LIN {X 0,Y 296.681,Z 512.231,A -85,B 0,C 180,E1 -16490.81,E2 -16490.81} C_VEL
LIN {X 0,Y 296.616,Z 512.901,A -85,B 0,C 180,E1 -16492.472,E2 -16492.472} C_VEL
LIN {X 0,Y 296.719,Z 512.686,A -85,B 0,C 180,E1 -16495.232,E2 -16495.232} C_VEL
LIN {X 0,Y 296.911,Z 511.914,A -85,B 0,C 180,E1 -16496.723,E2 -16496.723} C_VEL
LIN {X 0,Y 297.383,Z 509.725,A -85,B 0,C 180,E1 -16499.024,E2 -16499.024} C_VEL
LIN {X 0,Y 298.001,Z 506.45,A -85,B 0,C 180,E1 -16501.251,E2 -16501.251} C_VEL
LIN {X 0,Y 298.906,Z 501.771,A -85,B 0,C 180,E1 -16503.538,E2 -16503.538} C_VEL
LIN {X 0,Y 300.159,Z 495.578,A -85,B 0,C 180,E1 -16505.824,E2 -16505.824} C_VEL
LIN {X 0,Y 301.385,Z 489.056,A -85,B 0,C 180,E1 -16507.716,E2 -16507.716} C_VEL
LIN {X 0,Y 302.931,Z 480.785,A -85,B 0,C 180,E1 -16509.639,E2 -16509.639} C_VEL
LIN {X 0,Y 304.466,Z 471.668,A -85,B 0,C 180,E1 -16511.353,E2 -16511.353} C_VEL
LIN {X 0,Y 306.154,Z 461.176,A -85,B 0,C 180,E1 -16512.929,E2 -16512.929} C_VEL
LIN {X 0,Y 307.794,Z 449.247,A -85,B 0,C 180,E1 -16514.327,E2 -16514.327} C_VEL
LIN {X 0,Y 307.85,Z 445.631,A -85,B 0,C 180,E1 -16514.72,E2 -16514.72} C_VEL
LIN {X 0,Y 305.288,Z 433.549,A -85,B 0,C 180,E1 -16516.069,E2 -16516.069} C_VEL
LIN {X 0,Y 301.496,Z 421.211,A -85,B 0,C 180,E1 -16517.278,E2 -16517.278} C_VEL
LIN {X 0,Y 297.926,Z 411.655,A -85,B 0,C 180,E1 -16518.096,E2 -16518.096} C_VEL
LIN {X 0,Y 297.834,Z 411.063,A -85,B 0,C 180,E1 -16518.137,E2 -16518.137} C_VEL
LIN {X 0,Y 298.025,Z 408.055,A -85,B 0,C 180,E1 -16522.184,E2 -16522.184} C_VEL
LIN {X 0,Y 298.192,Z 405.628,A -85,B 0,C 180,E1 -16525.572,E2 -16525.572} C_VEL
LIN {X 0,Y 298.291,Z 403.444,A -85,B 0,C 180,E1 -16528.779,E2 -16528.779} C_VEL
LIN {X 0,Y 298.434,Z 403.312,A -85,B 0,C 180,E1 -16531.901,E2 -16531.901} C_VEL
LIN {X 0,Y 298.483,Z 403.308,A -85,B 0,C 180,E1 -16534.924,E2 -16534.924} C_VEL
LIN {X 0,Y 298.482,Z 403.306,A -85,B 0,C 180,E1 -16537.869,E2 -16537.869} C_VEL
LIN {X 0,Y 298.55,Z 403.298,A -85,B 0,C 180,E1 -16540.758,E2 -16540.758} C_VEL
LIN {X 0,Y 298.575,Z 403.294,A -85,B 0,C 180,E1 -16544.994,E2 -16544.994} C_VEL
LIN {X 0,Y 298.577,Z 403.292,A -85,B 0,C 180,E1 -16549.146,E2 -16549.146} C_VEL
LIN {X 0,Y 298.735,Z 403.271,A -85,B 0,C 180,E1 -16552.197,E2 -16552.197} C_VEL
LIN {X 0,Y 298.066,Z 403.353,A -85,B 0,C 180,E1 -16553.321,E2 -16553.321} C_VEL
LIN {X 0,Y 295.213,Z 403.713,A -85,B 0,C 180,E1 -16555.151,E2 -16555.151} C_VEL
LIN {X 0,Y 292.833,Z 404.01,A -85,B 0,C 180,E1 -16556.636,E2 -16556.636} C_VEL
LIN {X 0,Y 291.871,Z 404.129,A -85,B 0,C 180,E1 -16557.787,E2 -16557.787} C_VEL
LIN {X 0,Y 291.823,Z 404.132,A -85,B 0,C 180,E1 -16558.176,E2 -16558.176} C_VEL
LIN {X 0,Y 291.962,Z 404.118,A -85,B 0,C 180,E1 -16560,E2 -16560} C_VEL
LIN {X 0,Y 291.788,Z 404.139,A -85,B 0,C 180,E1 -16562.761,E2 -16562.761} C_VEL
LIN {X 0,Y 291.727,Z 404.147,A -85,B 0,C 180,E1 -16566.918,E2 -16566.918} C_VEL
LIN {X 0,Y 291.611,Z 404.161,A -85,B 0,C 180,E1 -16569.713,E2 -16569.713} C_VEL
LIN {X 0,Y 291.505,Z 404.175,A -85,B 0,C 180,E1 -16573.951,E2 -16573.951} C_VEL
LIN {X 0,Y 291.471,Z 404.181,A -85,B 0,C 180,E1 -16576.819,E2 -16576.819} C_VEL
LIN {X 0,Y 291.479,Z 404.18,A -85,B 0,C 180,E1 -16579.901,E2 -16579.901} C_VEL
LIN {X 0,Y 291.422,Z 404.189,A -85,B 0,C 180,E1 -16584.204,E2 -16584.204} C_VEL
LIN {X 0,Y 291.404,Z 404.192,A -85,B 0,C 180,E1 -16587.274,E2 -16587.274} C_VEL
LIN {X 0,Y 291.319,Z 404.202,A -85,B 0,C 180,E1 -16590.439,E2 -16590.439} C_VEL
LIN {X 0,Y 291.33,Z 404.198,A -85,B 0,C 180,E1 -16593.701,E2 -16593.701} C_VEL
LIN {X 0,Y 291.43,Z 404.372,A -85,B 0,C 180,E1 -16597.077,E2 -16597.077} C_VEL
LIN {X 0,Y 292.013,Z 407.676,A -85,B 0,C 180,E1 -16600.528,E2 -16600.528} C_VEL
LIN {X 0,Y 292.688,Z 411.501,A -85,B 0,C 180,E1 -16604.135,E2 -16604.135} C_VEL
LIN {X 0,Y 293.487,Z 415.946,A -85,B 0,C 180,E1 -16607.932,E2 -16607.932} C_VEL
LIN {X 0,Y 294.295,Z 420.631,A -85,B 0,C 180,E1 -16611.622,E2 -16611.622} C_VEL
LIN {X 0,Y 294.316,Z 423.007,A -85,B 0,C 180,E1 -16613.35,E2 -16613.35} C_VEL
LIN {X 0,Y 293.501,Z 427.798,A -85,B 0,C 180,E1 -16616.586,E2 -16616.586} C_VEL
LIN {X 0,Y 292.428,Z 433.947,A -85,B 0,C 180,E1 -16620.555,E2 -16620.555} C_VEL
LIN {X 0,Y 291.578,Z 439.819,A -85,B 0,C 180,E1 -16624.22,E2 -16624.22} C_VEL
LIN {X 0,Y 294.842,Z 453.988,A -85,B 0,C 180,E1 -16625.215,E2 -16625.215} C_VEL
LIN {X 0,Y 296.937,Z 466.347,A -85,B 0,C 180,E1 -16626.278,E2 -16626.278} C_VEL
LIN {X 0,Y 297.877,Z 477.919,A -85,B 0,C 180,E1 -16627.433,E2 -16627.433} C_VEL
LIN {X 0,Y 298.271,Z 489.026,A -85,B 0,C 180,E1 -16628.763,E2 -16628.763} C_VEL
LIN {X 0,Y 298.073,Z 493.023,A -85,B 0,C 180,E1 -16629.291,E2 -16629.291} C_VEL
LIN {X 0,Y 296.243,Z 503.418,A -85,B 0,C 180,E1 -16630.785,E2 -16630.785} C_VEL
LIN {X 0,Y 294.557,Z 512.927,A -85,B 0,C 180,E1 -16632.496,E2 -16632.496} C_VEL
LIN {X 0,Y 293.442,Z 519.865,A -85,B 0,C 180,E1 -16634.016,E2 -16634.016} C_VEL
LIN {X 0,Y 292.007,Z 527.627,A -85,B 0,C 180,E1 -16636.076,E2 -16636.076} C_VEL
LIN {X 0,Y 290.904,Z 533.892,A -85,B 0,C 180,E1 -16638.153,E2 -16638.153} C_VEL
LIN {X 0,Y 290.221,Z 538.898,A -85,B 0,C 180,E1 -16640.243,E2 -16640.243} C_VEL
LIN {X 0,Y 289.814,Z 542.782,A -85,B 0,C 180,E1 -16642.338,E2 -16642.338} C_VEL
LIN {X 0,Y 289.624,Z 545.643,A -85,B 0,C 180,E1 -16644.433,E2 -16644.433} C_VEL
LIN {X 0,Y 289.583,Z 547.008,A -85,B 0,C 180,E1 -16645.827,E2 -16645.827} C_VEL
LIN {X 0,Y 289.557,Z 547.975,A -85,B 0,C 180,E1 -16647.22,E2 -16647.22} C_VEL
LIN {X 0,Y 289.58,Z 548.533,A -85,B 0,C 180,E1 -16648.612,E2 -16648.612} C_VEL
LIN {X 0,Y 289.694,Z 548.659,A -85,B 0,C 180,E1 -16650.003,E2 -16650.003} C_VEL
LIN {X 0,Y 289.609,Z 548.378,A -85,B 0,C 180,E1 -16651.393,E2 -16651.393} C_VEL
LIN {X 0,Y 289.567,Z 547.706,A -85,B 0,C 180,E1 -16652.785,E2 -16652.785} C_VEL
LIN {X 0,Y 289.601,Z 546.628,A -85,B 0,C 180,E1 -16654.178,E2 -16654.178} C_VEL
LIN {X 0,Y 289.637,Z 544.779,A -85,B 0,C 180,E1 -16655.81,E2 -16655.81} C_VEL
LIN {X 0,Y 289.908,Z 540.719,A -85,B 0,C 180,E1 -16658.366,E2 -16658.366} C_VEL
LIN {X 0,Y 290.45,Z 536.166,A -85,B 0,C 180,E1 -16660.458,E2 -16660.458} C_VEL
LIN {X 0,Y 291.383,Z 529.252,A -85,B 0,C 180,E1 -16662.894,E2 -16662.894} C_VEL
LIN {X 0,Y 292.59,Z 521.762,A -85,B 0,C 180,E1 -16664.967,E2 -16664.967} C_VEL
LIN {X 0,Y 293.871,Z 514.132,A -85,B 0,C 180,E1 -16666.68,E2 -16666.68} C_VEL
LIN {X 0,Y 295.154,Z 504.871,A -85,B 0,C 180,E1 -16668.393,E2 -16668.393} C_VEL
LIN {X 0,Y 296.846,Z 494.612,A -85,B 0,C 180,E1 -16669.9,E2 -16669.9} C_VEL
LIN {X 0,Y 297.487,Z 489.241,A -85,B 0,C 180,E1 -16670.576,E2 -16670.576} C_VEL
LIN {X 0,Y 296.781,Z 477.347,A -85,B 0,C 180,E1 -16671.956,E2 -16671.956} C_VEL
LIN {X 0,Y 295.703,Z 465.945,A -85,B 0,C 180,E1 -16673.033,E2 -16673.033} C_VEL
LIN {X 0,Y 293.736,Z 453.233,A -85,B 0,C 180,E1 -16674.003,E2 -16674.003} C_VEL
LIN {X 0,Y 291.321,Z 441.044,A -85,B 0,C 180,E1 -16674.724,E2 -16674.724} C_VEL
LIN {X 0,Y 292.187,Z 434.465,A -85,B 0,C 180,E1 -16678.757,E2 -16678.757} C_VEL
LIN {X 0,Y 293.285,Z 427.694,A -85,B 0,C 180,E1 -16682.996,E2 -16682.996} C_VEL
LIN {X 0,Y 294.052,Z 423.605,A -85,B 0,C 180,E1 -16685.647,E2 -16685.647} C_VEL
LIN {X 0,Y 294.158,Z 420.178,A -85,B 0,C 180,E1 -16687.96,E2 -16687.96} C_VEL
LIN {X 0,Y 293.255,Z 414.608,A -85,B 0,C 180,E1 -16692.018,E2 -16692.018} C_VEL
LIN {X 0,Y 292.387,Z 409.776,A -85,B 0,C 180,E1 -16695.808,E2 -16695.808} C_VEL
LIN {X 0,Y 291.492,Z 404.752,A -85,B 0,C 180,E1 -16700.024,E2 -16700.024} C_VEL
LIN {X 0,Y 291.369,Z 404.193,A -85,B 0,C 180,E1 -16700.524,E2 -16700.524} C_VEL
LIN {X 0,Y 291.415,Z 404.187,A -85,B 0,C 180,E1 -16702.92,E2 -16702.92} C_VEL
LIN {X 0,Y 291.352,Z 404.194,A -85,B 0,C 180,E1 -16706.302,E2 -16706.302} C_VEL
LIN {X 0,Y 291.391,Z 404.189,A -85,B 0,C 180,E1 -16710.262,E2 -16710.262} C_VEL
LIN {X 0,Y 291.42,Z 404.185,A -85,B 0,C 180,E1 -16714.272,E2 -16714.272} C_VEL
LIN {X 0,Y 291.389,Z 404.186,A -85,B 0,C 180,E1 -16717.3,E2 -16717.3} C_VEL
LIN {X 0,Y 291.466,Z 404.181,A -85,B 0,C 180,E1 -16720.271,E2 -16720.271} C_VEL
LIN {X 0,Y 291.549,Z 404.171,A -85,B 0,C 180,E1 -16724.635,E2 -16724.635} C_VEL
LIN {X 0,Y 291.543,Z 404.169,A -85,B 0,C 180,E1 -16728.881,E2 -16728.881} C_VEL
LIN {X 0,Y 291.695,Z 404.15,A -85,B 0,C 180,E1 -16731.688,E2 -16731.688} C_VEL
LIN {X 0,Y 291.632,Z 404.159,A -85,B 0,C 180,E1 -16734.468,E2 -16734.468} C_VEL
LIN {X 0,Y 291.895,Z 404.124,A -85,B 0,C 180,E1 -16738.62,E2 -16738.62} C_VEL
LIN {X 0,Y 291.895,Z 404.123,A -85,B 0,C 180,E1 -16741.38,E2 -16741.38} C_VEL
LIN {X 0,Y 291.753,Z 404.129,A -85,B 0,C 180,E1 -16746.918,E2 -16746.918} C_VEL
LIN {X 0,Y 291.637,Z 404.153,A -85,B 0,C 180,E1 -16749.712,E2 -16749.712} C_VEL
LIN {X 0,Y 291.529,Z 404.172,A -85,B 0,C 180,E1 -16753.95,E2 -16753.95} C_VEL
LIN {X 0,Y 291.494,Z 404.17,A -85,B 0,C 180,E1 -16756.817,E2 -16756.817} C_VEL
LIN {X 0,Y 291.459,Z 404.17,A -85,B 0,C 180,E1 -16759.874,E2 -16759.874} C_VEL
LIN {X 0,Y 291.408,Z 404.183,A -85,B 0,C 180,E1 -16764.205,E2 -16764.205} C_VEL
LIN {X 0,Y 291.427,Z 404.184,A -85,B 0,C 180,E1 -16767.271,E2 -16767.271} C_VEL
LIN {X 0,Y 291.341,Z 404.188,A -85,B 0,C 180,E1 -16770.436,E2 -16770.436} C_VEL
LIN {X 0,Y 291.351,Z 404.188,A -85,B 0,C 180,E1 -16773.697,E2 -16773.697} C_VEL
LIN {X 0,Y 291.379,Z 404.19,A -85,B 0,C 180,E1 -16777.252,E2 -16777.252} C_VEL
LIN {X 0,Y 291.34,Z 404.192,A -85,B 0,C 180,E1 -16780.641,E2 -16780.641} C_VEL
LIN {X 0,Y 291.32,Z 404.188,A -85,B 0,C 180,E1 -16784.396,E2 -16784.396} C_VEL
LIN {X 0,Y 291.333,Z 404.193,A -85,B 0,C 180,E1 -16788.403,E2 -16788.403} C_VEL
LIN {X 0,Y 291.354,Z 404.19,A -85,B 0,C 180,E1 -16791.156,E2 -16791.156} C_VEL
LIN {X 0,Y 291.367,Z 404.189,A -85,B 0,C 180,E1 -16794.624,E2 -16794.624} C_VEL
LIN {X 0,Y 291.376,Z 404.188,A -85,B 0,C 180,E1 -16797.949,E2 -16797.949} C_VEL
LIN {X 0,Y 291.383,Z 404.191,A -85,B 0,C 180,E1 -16801.156,E2 -16801.156} C_VEL
LIN {X 0,Y 291.418,Z 404.185,A -85,B 0,C 180,E1 -16804.27,E2 -16804.27} C_VEL
LIN {X 0,Y 291.387,Z 404.188,A -85,B 0,C 180,E1 -16807.298,E2 -16807.298} C_VEL
LIN {X 0,Y 291.463,Z 404.179,A -85,B 0,C 180,E1 -16810.268,E2 -16810.268} C_VEL
LIN {X 0,Y 291.544,Z 404.171,A -85,B 0,C 180,E1 -16814.632,E2 -16814.632} C_VEL
LIN {X 0,Y 291.413,Z 404.184,A -85,B 0,C 180,E1 -16817.462,E2 -16817.462} C_VEL
LIN {X 0,Y 291.24,Z 404.209,A -85,B 0,C 180,E1 -16820.273,E2 -16820.273} C_VEL
LIN {X 0,Y 291.175,Z 404.529,A -85,B 0,C 180,E1 -16821.731,E2 -16821.731} C_VEL
LIN {X 0,Y 291.222,Z 406.671,A -85,B 0,C 180,E1 -16824.458,E2 -16824.458} C_VEL
LIN {X 0,Y 290.562,Z 409.89,A -85,B 0,C 180,E1 -16828.438,E2 -16828.438} C_VEL
LIN {X 0,Y 294.972,Z 424.125,A -85,B 0,C 180,E1 -16829.537,E2 -16829.537} C_VEL
LIN {X 0,Y 297.721,Z 434.159,A -85,B 0,C 180,E1 -16830.483,E2 -16830.483} C_VEL
LIN {X 0,Y 299.896,Z 445.157,A -85,B 0,C 180,E1 -16831.676,E2 -16831.676} C_VEL
LIN {X 0,Y 298.681,Z 455.984,A -85,B 0,C 180,E1 -16832.863,E2 -16832.863} C_VEL
LIN {X 0,Y 297.212,Z 466.632,A -85,B 0,C 180,E1 -16834.335,E2 -16834.335} C_VEL
LIN {X 0,Y 295.569,Z 477.057,A -85,B 0,C 180,E1 -16836.14,E2 -16836.14} C_VEL
LIN {X 0,Y 294.202,Z 485.218,A -85,B 0,C 180,E1 -16837.892,E2 -16837.892} C_VEL
LIN {X 0,Y 293.014,Z 491.971,A -85,B 0,C 180,E1 -16839.663,E2 -16839.663} C_VEL
LIN {X 0,Y 291.926,Z 498.542,A -85,B 0,C 180,E1 -16841.805,E2 -16841.805} C_VEL
LIN {X 0,Y 291.052,Z 503.752,A -85,B 0,C 180,E1 -16843.97,E2 -16843.97} C_VEL
LIN {X 0,Y 290.419,Z 507.763,A -85,B 0,C 180,E1 -16846.155,E2 -16846.155} C_VEL
LIN {X 0,Y 289.832,Z 511.314,A -85,B 0,C 180,E1 -16848.969,E2 -16848.969} C_VEL
LIN {X 0,Y 289.554,Z 512.957,A -85,B 0,C 180,E1 -16851.347,E2 -16851.347} C_VEL
LIN {X 0,Y 289.519,Z 513.386,A -85,B 0,C 180,E1 -16852.851,E2 -16852.851} C_VEL
LIN {X 0,Y 289.572,Z 513.384,A -85,B 0,C 180,E1 -16854.364,E2 -16854.364} C_VEL
LIN {X 0,Y 289.755,Z 512.734,A -85,B 0,C 180,E1 -16856.177,E2 -16856.177} C_VEL
LIN {X 0,Y 290.291,Z 510.467,A -85,B 0,C 180,E1 -16858.957,E2 -16858.957} C_VEL
LIN {X 0,Y 290.957,Z 507.246,A -85,B 0,C 180,E1 -16861.283,E2 -16861.283} C_VEL
LIN {X 0,Y 291.87,Z 502.682,A -85,B 0,C 180,E1 -16863.626,E2 -16863.626} C_VEL
LIN {X 0,Y 293.114,Z 496.848,A -85,B 0,C 180,E1 -16865.886,E2 -16865.886} C_VEL
LIN {X 0,Y 294.559,Z 489.677,A -85,B 0,C 180,E1 -16868.061,E2 -16868.061} C_VEL
LIN {X 0,Y 296.268,Z 480.874,A -85,B 0,C 180,E1 -16870.146,E2 -16870.146} C_VEL
LIN {X 0,Y 298.012,Z 471.092,A -85,B 0,C 180,E1 -16871.998,E2 -16871.998} C_VEL
LIN {X 0,Y 299.664,Z 461.06,A -85,B 0,C 180,E1 -16873.502,E2 -16873.502} C_VEL
LIN {X 0,Y 301.294,Z 449.764,A -85,B 0,C 180,E1 -16874.846,E2 -16874.846} C_VEL
LIN {X 0,Y 301.051,Z 445.998,A -85,B 0,C 180,E1 -16875.293,E2 -16875.293} C_VEL
LIN {X 0,Y 298.548,Z 434.444,A -85,B 0,C 180,E1 -16876.638,E2 -16876.638} C_VEL
LIN {X 0,Y 294.976,Z 422.795,A -85,B 0,C 180,E1 -16877.84,E2 -16877.84} C_VEL
LIN {X 0,Y 290.933,Z 412.057,A -85,B 0,C 180,E1 -16878.81,E2 -16878.81} C_VEL
LIN {X 0,Y 290.844,Z 411.521,A -85,B 0,C 180,E1 -16878.875,E2 -16878.875} C_VEL
LIN {X 0,Y 291.05,Z 408.634,A -85,B 0,C 180,E1 -16882.866,E2 -16882.866} C_VEL
LIN {X 0,Y 291.196,Z 406.275,A -85,B 0,C 180,E1 -16886.282,E2 -16886.282} C_VEL
LIN {X 0,Y 291.268,Z 404.208,A -85,B 0,C 180,E1 -16889.555,E2 -16889.555} C_VEL
LIN {X 0,Y 291.423,Z 404.186,A -85,B 0,C 180,E1 -16893.155,E2 -16893.155} C_VEL
LIN {X 0,Y 291.436,Z 404.186,A -85,B 0,C 180,E1 -16897.304,E2 -16897.304} C_VEL
LIN {X 0,Y 291.497,Z 404.175,A -85,B 0,C 180,E1 -16900.273,E2 -16900.273} C_VEL
LIN {X 0,Y 291.522,Z 404.17,A -85,B 0,C 180,E1 -16904.634,E2 -16904.634} C_VEL
LIN {X 0,Y 291.52,Z 404.172,A -85,B 0,C 180,E1 -16908.88,E2 -16908.88} C_VEL
LIN {X 0,Y 291.685,Z 404.148,A -85,B 0,C 180,E1 -16912.201,E2 -16912.201} C_VEL
LIN {X 0,Y 291.773,Z 404.141,A -85,B 0,C 180,E1 -16917.239,E2 -16917.239} C_VEL
LIN {X 0,Y 291.823,Z 404.132,A -85,B 0,C 180,E1 -16918.176,E2 -16918.176} C_VEL
LIN {X 0,Y 291.206,Z 404.212,A -85,B 0,C 180,E1 -16919.329,E2 -16919.329} C_VEL
LIN {X 0,Y 288.248,Z 404.587,A -85,B 0,C 180,E1 -16921.201,E2 -16921.201} C_VEL
LIN {X 0,Y 285.69,Z 404.905,A -85,B 0,C 180,E1 -16922.722,E2 -16922.722} C_VEL
LIN {X 0,Y 284.59,Z 405.037,A -85,B 0,C 180,E1 -16923.904,E2 -16923.904} C_VEL
LIN {X 0,Y 284.504,Z 405.045,A -85,B 0,C 180,E1 -16924.305,E2 -16924.305} C_VEL
LIN {X 0,Y 284.679,Z 405.025,A -85,B 0,C 180,E1 -16927.091,E2 -16927.091} C_VEL
LIN {X 0,Y 284.549,Z 405.042,A -85,B 0,C 180,E1 -16929.956,E2 -16929.956} C_VEL
LIN {X 0,Y 284.464,Z 405.052,A -85,B 0,C 180,E1 -16934.304,E2 -16934.304} C_VEL
LIN {X 0,Y 284.412,Z 405.058,A -85,B 0,C 180,E1 -16937.249,E2 -16937.249} C_VEL
LIN {X 0,Y 284.411,Z 405.059,A -85,B 0,C 180,E1 -16940.24,E2 -16940.24} C_VEL
LIN {X 0,Y 284.385,Z 405.066,A -85,B 0,C 180,E1 -16943.891,E2 -16943.891} C_VEL
LIN {X 0,Y 284.313,Z 405.076,A -85,B 0,C 180,E1 -16948.013,E2 -16948.013} C_VEL
LIN {X 0,Y 284.278,Z 405.078,A -85,B 0,C 180,E1 -16951.277,E2 -16951.277} C_VEL
LIN {X 0,Y 284.334,Z 405.068,A -85,B 0,C 180,E1 -16955.805,E2 -16955.805} C_VEL
LIN {X 0,Y 284.653,Z 406.913,A -85,B 0,C 180,E1 -16958.115,E2 -16958.115} C_VEL
LIN {X 0,Y 285.281,Z 410.368,A -85,B 0,C 180,E1 -16961.695,E2 -16961.695} C_VEL
LIN {X 0,Y 285.991,Z 414.396,A -85,B 0,C 180,E1 -16965.451,E2 -16965.451} C_VEL
LIN {X 0,Y 286.83,Z 419.085,A -85,B 0,C 180,E1 -16969.427,E2 -16969.427} C_VEL
LIN {X 0,Y 287.326,Z 422.758,A -85,B 0,C 180,E1 -16972.306,E2 -16972.306} C_VEL
LIN {X 0,Y 286.95,Z 426.313,A -85,B 0,C 180,E1 -16974.865,E2 -16974.865} C_VEL
LIN {X 0,Y 285.649,Z 433.115,A -85,B 0,C 180,E1 -16979.444,E2 -16979.444} C_VEL
LIN {X 0,Y 284.685,Z 439.351,A -85,B 0,C 180,E1 -16983.471,E2 -16983.471} C_VEL
LIN {X 0,Y 287.348,Z 450.529,A -85,B 0,C 180,E1 -16984.276,E2 -16984.276} C_VEL
LIN {X 0,Y 289.767,Z 463.231,A -85,B 0,C 180,E1 -16985.37,E2 -16985.37} C_VEL
LIN {X 0,Y 291.055,Z 475.183,A -85,B 0,C 180,E1 -16986.574,E2 -16986.574} C_VEL
LIN {X 0,Y 291.496,Z 487.557,A -85,B 0,C 180,E1 -16988.059,E2 -16988.059} C_VEL
LIN {X 0,Y 291.227,Z 494.231,A -85,B 0,C 180,E1 -16988.966,E2 -16988.966} C_VEL
LIN {X 0,Y 289.334,Z 504.284,A -85,B 0,C 180,E1 -16990.492,E2 -16990.492} C_VEL
LIN {X 0,Y 287.645,Z 513.364,A -85,B 0,C 180,E1 -16992.208,E2 -16992.208} C_VEL
LIN {X 0,Y 286.302,Z 520.998,A -85,B 0,C 180,E1 -16993.972,E2 -16993.972} C_VEL
LIN {X 0,Y 284.863,Z 528.465,A -85,B 0,C 180,E1 -16996.084,E2 -16996.084} C_VEL
LIN {X 0,Y 283.668,Z 535.378,A -85,B 0,C 180,E1 -16998.571,E2 -16998.571} C_VEL
LIN {X 0,Y 282.999,Z 539.967,A -85,B 0,C 180,E1 -17000.714,E2 -17000.714} C_VEL
LIN {X 0,Y 282.679,Z 543.485,A -85,B 0,C 180,E1 -17002.862,E2 -17002.862} C_VEL
LIN {X 0,Y 282.562,Z 545.249,A -85,B 0,C 180,E1 -17004.293,E2 -17004.293} C_VEL
LIN {X 0,Y 282.502,Z 546.606,A -85,B 0,C 180,E1 -17005.723,E2 -17005.723} C_VEL
LIN {X 0,Y 282.483,Z 547.565,A -85,B 0,C 180,E1 -17007.151,E2 -17007.151} C_VEL
LIN {X 0,Y 282.495,Z 548.106,A -85,B 0,C 180,E1 -17008.577,E2 -17008.577} C_VEL
LIN {X 0,Y 282.606,Z 548.222,A -85,B 0,C 180,E1 -17010.003,E2 -17010.003} C_VEL
LIN {X 0,Y 282.522,Z 547.933,A -85,B 0,C 180,E1 -17011.428,E2 -17011.428} C_VEL
LIN {X 0,Y 282.493,Z 547.253,A -85,B 0,C 180,E1 -17012.855,E2 -17012.855} C_VEL
LIN {X 0,Y 282.519,Z 546.157,A -85,B 0,C 180,E1 -17014.283,E2 -17014.283} C_VEL
LIN {X 0,Y 282.56,Z 544.512,A -85,B 0,C 180,E1 -17015.785,E2 -17015.785} C_VEL
LIN {X 0,Y 282.742,Z 541.471,A -85,B 0,C 180,E1 -17017.86,E2 -17017.86} C_VEL
LIN {X 0,Y 283.218,Z 537.27,A -85,B 0,C 180,E1 -17020.006,E2 -17020.006} C_VEL
LIN {X 0,Y 284.073,Z 530.861,A -85,B 0,C 180,E1 -17022.505,E2 -17022.505} C_VEL
LIN {X 0,Y 285.3,Z 523.891,A -85,B 0,C 180,E1 -17024.628,E2 -17024.628} C_VEL
LIN {X 0,Y 286.772,Z 515.147,A -85,B 0,C 180,E1 -17026.738,E2 -17026.738} C_VEL
LIN {X 0,Y 288.073,Z 506.18,A -85,B 0,C 180,E1 -17028.493,E2 -17028.493} C_VEL
LIN {X 0,Y 289.793,Z 496.377,A -85,B 0,C 180,E1 -17030.035,E2 -17030.035} C_VEL
LIN {X 0,Y 290.597,Z 489.898,A -85,B 0,C 180,E1 -17030.902,E2 -17030.902} C_VEL
LIN {X 0,Y 289.937,Z 477.916,A -85,B 0,C 180,E1 -17032.347,E2 -17032.347} C_VEL
LIN {X 0,Y 288.783,Z 465.662,A -85,B 0,C 180,E1 -17033.548,E2 -17033.548} C_VEL
LIN {X 0,Y 286.787,Z 452.711,A -85,B 0,C 180,E1 -17034.567,E2 -17034.567} C_VEL
LIN {X 0,Y 284.34,Z 440.617,A -85,B 0,C 180,E1 -17035.332,E2 -17035.332} C_VEL
LIN {X 0,Y 285.115,Z 435.209,A -85,B 0,C 180,E1 -17038.732,E2 -17038.732} C_VEL
LIN {X 0,Y 286.12,Z 429.035,A -85,B 0,C 180,E1 -17042.713,E2 -17042.713} C_VEL
LIN {X 0,Y 287.065,Z 423.909,A -85,B 0,C 180,E1 -17046.107,E2 -17046.107} C_VEL
LIN {X 0,Y 287.086,Z 420.599,A -85,B 0,C 180,E1 -17048.429,E2 -17048.429} C_VEL
LIN {X 0,Y 286.156,Z 415.15,A -85,B 0,C 180,E1 -17052.54,E2 -17052.54} C_VEL
LIN {X 0,Y 285.268,Z 410.395,A -85,B 0,C 180,E1 -17056.384,E2 -17056.384} C_VEL
LIN {X 0,Y 284.541,Z 406.147,A -85,B 0,C 180,E1 -17060.045,E2 -17060.045} C_VEL
LIN {X 0,Y 284.316,Z 405.071,A -85,B 0,C 180,E1 -17061.153,E2 -17061.153} C_VEL
LIN {X 0,Y 284.349,Z 405.067,A -85,B 0,C 180,E1 -17064.653,E2 -17064.653} C_VEL
LIN {X 0,Y 284.301,Z 405.075,A -85,B 0,C 180,E1 -17068.726,E2 -17068.726} C_VEL
LIN {X 0,Y 284.402,Z 405.059,A -85,B 0,C 180,E1 -17072.828,E2 -17072.828} C_VEL
LIN {X 0,Y 284.374,Z 405.064,A -85,B 0,C 180,E1 -17076.707,E2 -17076.707} C_VEL
LIN {X 0,Y 284.411,Z 405.057,A -85,B 0,C 180,E1 -17081.262,E2 -17081.262} C_VEL
LIN {X 0,Y 284.486,Z 405.052,A -85,B 0,C 180,E1 -17084.47,E2 -17084.47} C_VEL
LIN {X 0,Y 284.495,Z 405.049,A -85,B 0,C 180,E1 -17088.602,E2 -17088.602} C_VEL
LIN {X 0,Y 284.647,Z 405.027,A -85,B 0,C 180,E1 -17091.481,E2 -17091.481} C_VEL
LIN {X 0,Y 284.603,Z 405.036,A -85,B 0,C 180,E1 -17094.331,E2 -17094.331} C_VEL
LIN {X 0,Y 284.861,Z 405,A -85,B 0,C 180,E1 -17098.586,E2 -17098.586} C_VEL
LIN {X 0,Y 284.861,Z 405,A -85,B 0,C 180,E1 -17101.414,E2 -17101.414} C_VEL
LIN {X 0,Y 284.705,Z 405.006,A -85,B 0,C 180,E1 -17107.09,E2 -17107.09} C_VEL
LIN {X 0,Y 284.574,Z 405.034,A -85,B 0,C 180,E1 -17109.955,E2 -17109.955} C_VEL
LIN {X 0,Y 284.486,Z 405.047,A -85,B 0,C 180,E1 -17114.302,E2 -17114.302} C_VEL
LIN {X 0,Y 284.433,Z 405.051,A -85,B 0,C 180,E1 -17117.248,E2 -17117.248} C_VEL
LIN {X 0,Y 284.387,Z 405.048,A -85,B 0,C 180,E1 -17120.242,E2 -17120.242} C_VEL
LIN {X 0,Y 284.377,Z 405.061,A -85,B 0,C 180,E1 -17123.874,E2 -17123.874} C_VEL
LIN {X 0,Y 284.403,Z 405.058,A -85,B 0,C 180,E1 -17127.172,E2 -17127.172} C_VEL
LIN {X 0,Y 284.301,Z 405.066,A -85,B 0,C 180,E1 -17131.274,E2 -17131.274} C_VEL
LIN {X 0,Y 284.348,Z 405.062,A -85,B 0,C 180,E1 -17135.347,E2 -17135.347} C_VEL
LIN {X 0,Y 284.315,Z 405.067,A -85,B 0,C 180,E1 -17138.168,E2 -17138.168} C_VEL
LIN {X 0,Y 284.276,Z 405.067,A -85,B 0,C 180,E1 -17142.123,E2 -17142.123} C_VEL
LIN {X 0,Y 284.275,Z 405.07,A -85,B 0,C 180,E1 -17146.19,E2 -17146.19} C_VEL
LIN {X 0,Y 284.313,Z 405.066,A -85,B 0,C 180,E1 -17150.022,E2 -17150.022} C_VEL
LIN {X 0,Y 284.337,Z 405.064,A -85,B 0,C 180,E1 -17153.612,E2 -17153.612} C_VEL
LIN {X 0,Y 284.313,Z 405.071,A -85,B 0,C 180,E1 -17157.188,E2 -17157.188} C_VEL
LIN {X 0,Y 284.361,Z 405.059,A -85,B 0,C 180,E1 -17160.374,E2 -17160.374} C_VEL
LIN {X 0,Y 284.38,Z 405.061,A -85,B 0,C 180,E1 -17163.584,E2 -17163.584} C_VEL
LIN {X 0,Y 284.372,Z 405.062,A -85,B 0,C 180,E1 -17166.705,E2 -17166.705} C_VEL
LIN {X 0,Y 284.408,Z 405.056,A -85,B 0,C 180,E1 -17171.259,E2 -17171.259} C_VEL
LIN {X 0,Y 284.482,Z 405.05,A -85,B 0,C 180,E1 -17174.467,E2 -17174.467} C_VEL
LIN {X 0,Y 284.395,Z 405.059,A -85,B 0,C 180,E1 -17177.147,E2 -17177.147} C_VEL
LIN {X 0,Y 284.197,Z 405.085,A -85,B 0,C 180,E1 -17180.029,E2 -17180.029} C_VEL
LIN {X 0,Y 284.147,Z 405.422,A -85,B 0,C 180,E1 -17181.63,E2 -17181.63} C_VEL
LIN {X 0,Y 284.182,Z 407.488,A -85,B 0,C 180,E1 -17184.32,E2 -17184.32} C_VEL
LIN {X 0,Y 283.6,Z 410.547,A -85,B 0,C 180,E1 -17187.867,E2 -17187.867} C_VEL
LIN {X 0,Y 287.779,Z 423.859,A -85,B 0,C 180,E1 -17188.923,E2 -17188.923} C_VEL
LIN {X 0,Y 291.167,Z 436.144,A -85,B 0,C 180,E1 -17190.128,E2 -17190.128} C_VEL
LIN {X 0,Y 292.955,Z 445.605,A -85,B 0,C 180,E1 -17191.195,E2 -17191.195} C_VEL
LIN {X 0,Y 292.938,Z 448.73,A -85,B 0,C 180,E1 -17191.544,E2 -17191.544} C_VEL
LIN {X 0,Y 291.45,Z 460.262,A -85,B 0,C 180,E1 -17192.935,E2 -17192.935} C_VEL
LIN {X 0,Y 289.987,Z 469.937,A -85,B 0,C 180,E1 -17194.393,E2 -17194.393} C_VEL
LIN {X 0,Y 288.606,Z 478.318,A -85,B 0,C 180,E1 -17195.938,E2 -17195.938} C_VEL
LIN {X 0,Y 287.204,Z 486.314,A -85,B 0,C 180,E1 -17197.732,E2 -17197.732} C_VEL
LIN {X 0,Y 285.811,Z 494.104,A -85,B 0,C 180,E1 -17199.909,E2 -17199.909} C_VEL
LIN {X 0,Y 284.696,Z 500.354,A -85,B 0,C 180,E1 -17202.109,E2 -17202.109} C_VEL
LIN {X 0,Y 283.863,Z 505.277,A -85,B 0,C 180,E1 -17204.331,E2 -17204.331} C_VEL
LIN {X 0,Y 283.221,Z 509.028,A -85,B 0,C 180,E1 -17206.578,E2 -17206.578} C_VEL
LIN {X 0,Y 282.724,Z 511.952,A -85,B 0,C 180,E1 -17209.159,E2 -17209.159} C_VEL
LIN {X 0,Y 282.44,Z 513.594,A -85,B 0,C 180,E1 -17211.913,E2 -17211.913} C_VEL
LIN {X 0,Y 282.437,Z 513.895,A -85,B 0,C 180,E1 -17213.458,E2 -17213.458} C_VEL
LIN {X 0,Y 282.521,Z 513.685,A -85,B 0,C 180,E1 -17215.014,E2 -17215.014} C_VEL
LIN {X 0,Y 282.717,Z 513.027,A -85,B 0,C 180,E1 -17216.577,E2 -17216.577} C_VEL
LIN {X 0,Y 283.022,Z 511.893,A -85,B 0,C 180,E1 -17218.148,E2 -17218.148} C_VEL
LIN {X 0,Y 283.659,Z 509.193,A -85,B 0,C 180,E1 -17220.52,E2 -17220.52} C_VEL
LIN {X 0,Y 284.452,Z 505.215,A -85,B 0,C 180,E1 -17222.922,E2 -17222.922} C_VEL
LIN {X 0,Y 285.582,Z 500.218,A -85,B 0,C 180,E1 -17225.161,E2 -17225.161} C_VEL
LIN {X 0,Y 286.909,Z 494.06,A -85,B 0,C 180,E1 -17227.316,E2 -17227.316} C_VEL
LIN {X 0,Y 288.454,Z 486.932,A -85,B 0,C 180,E1 -17229.302,E2 -17229.302} C_VEL
LIN {X 0,Y 290.221,Z 477.718,A -85,B 0,C 180,E1 -17231.349,E2 -17231.349} C_VEL
LIN {X 0,Y 292.05,Z 468.053,A -85,B 0,C 180,E1 -17233.06,E2 -17233.06} C_VEL
LIN {X 0,Y 293.594,Z 458.467,A -85,B 0,C 180,E1 -17234.437,E2 -17234.437} C_VEL
LIN {X 0,Y 294.798,Z 449.462,A -85,B 0,C 180,E1 -17235.495,E2 -17235.495} C_VEL
LIN {X 0,Y 292.696,Z 438.628,A -85,B 0,C 180,E1 -17236.857,E2 -17236.857} C_VEL
LIN {X 0,Y 289.25,Z 426.705,A -85,B 0,C 180,E1 -17238.184,E2 -17238.184} C_VEL
LIN {X 0,Y 284.877,Z 415.028,A -85,B 0,C 180,E1 -17239.349,E2 -17239.349} C_VEL
LIN {X 0,Y 283.821,Z 412.012,A -85,B 0,C 180,E1 -17239.633,E2 -17239.633} C_VEL
LIN {X 0,Y 284.049,Z 409.242,A -85,B 0,C 180,E1 -17243.572,E2 -17243.572} C_VEL
LIN {X 0,Y 284.237,Z 406.801,A -85,B 0,C 180,E1 -17247.205,E2 -17247.205} C_VEL
LIN {X 0,Y 284.252,Z 405.081,A -85,B 0,C 180,E1 -17249.916,E2 -17249.916} C_VEL
LIN {X 0,Y 284.364,Z 405.066,A -85,B 0,C 180,E1 -17253.585,E2 -17253.585} C_VEL
LIN {X 0,Y 284.388,Z 405.064,A -85,B 0,C 180,E1 -17256.709,E2 -17256.709} C_VEL
LIN {X 0,Y 284.419,Z 405.055,A -85,B 0,C 180,E1 -17259.87,E2 -17259.87} C_VEL
LIN {X 0,Y 284.46,Z 405.049,A -85,B 0,C 180,E1 -17264.469,E2 -17264.469} C_VEL
LIN {X 0,Y 284.471,Z 405.052,A -85,B 0,C 180,E1 -17268.601,E2 -17268.601} C_VEL
LIN {X 0,Y 284.641,Z 405.031,A -85,B 0,C 180,E1 -17271.481,E2 -17271.481} C_VEL
LIN {X 0,Y 284.586,Z 405.037,A -85,B 0,C 180,E1 -17274.331,E2 -17274.331} C_VEL
LIN {X 0,Y 284.84,Z 405.004,A -85,B 0,C 180,E1 -17278.586,E2 -17278.586} C_VEL
LIN {X 0,Y 284.843,Z 405.005,A -85,B 0,C 180,E1 -17281.414,E2 -17281.414} C_VEL
LIN {X 0,Y 284.504,Z 405.045,A -85,B 0,C 180,E1 -17284.305,E2 -17284.305} C_VEL
LIN {X 0,Y 283.857,Z 405.127,A -85,B 0,C 180,E1 -17285.488,E2 -17285.488} C_VEL
LIN {X 0,Y 281.053,Z 405.476,A -85,B 0,C 180,E1 -17287.415,E2 -17287.415} C_VEL
LIN {X 0,Y 278.638,Z 405.779,A -85,B 0,C 180,E1 -17288.98,E2 -17288.98} C_VEL
LIN {X 0,Y 277.562,Z 405.913,A -85,B 0,C 180,E1 -17290.192,E2 -17290.192} C_VEL
LIN {X 0,Y 277.452,Z 405.924,A -85,B 0,C 180,E1 -17290.603,E2 -17290.603} C_VEL
LIN {X 0,Y 277.417,Z 405.93,A -85,B 0,C 180,E1 -17294.675,E2 -17294.675} C_VEL
LIN {X 0,Y 277.36,Z 405.938,A -85,B 0,C 180,E1 -17299.233,E2 -17299.233} C_VEL
LIN {X 0,Y 277.365,Z 405.941,A -85,B 0,C 180,E1 -17303.917,E2 -17303.917} C_VEL
LIN {X 0,Y 277.308,Z 405.947,A -85,B 0,C 180,E1 -17307.506,E2 -17307.506} C_VEL
LIN {X 0,Y 277.257,Z 405.954,A -85,B 0,C 180,E1 -17310.483,E2 -17310.483} C_VEL
LIN {X 0,Y 277.303,Z 406.009,A -85,B 0,C 180,E1 -17315.21,E2 -17315.21} C_VEL
LIN {X 0,Y 277.885,Z 409.507,A -85,B 0,C 180,E1 -17319.219,E2 -17319.219} C_VEL
LIN {X 0,Y 278.581,Z 413.17,A -85,B 0,C 180,E1 -17322.984,E2 -17322.984} C_VEL
LIN {X 0,Y 279.389,Z 417.772,A -85,B 0,C 180,E1 -17327.225,E2 -17327.225} C_VEL
LIN {X 0,Y 280.216,Z 422.478,A -85,B 0,C 180,E1 -17331.174,E2 -17331.174} C_VEL
LIN {X 0,Y 280.253,Z 425.345,A -85,B 0,C 180,E1 -17333.367,E2 -17333.367} C_VEL
LIN {X 0,Y 279.436,Z 429.605,A -85,B 0,C 180,E1 -17336.409,E2 -17336.409} C_VEL
LIN {X 0,Y 278.309,Z 435.622,A -85,B 0,C 180,E1 -17340.504,E2 -17340.504} C_VEL
LIN {X 0,Y 277.77,Z 438.862,A -85,B 0,C 180,E1 -17342.667,E2 -17342.667} C_VEL
LIN {X 0,Y 281.308,Z 453.467,A -85,B 0,C 180,E1 -17343.817,E2 -17343.817} C_VEL
LIN {X 0,Y 283.391,Z 465.534,A -85,B 0,C 180,E1 -17344.945,E2 -17344.945} C_VEL
LIN {X 0,Y 284.434,Z 476.24,A -85,B 0,C 180,E1 -17346.096,E2 -17346.096} C_VEL
LIN {X 0,Y 284.782,Z 488.96,A -85,B 0,C 180,E1 -17347.705,E2 -17347.705} C_VEL
LIN {X 0,Y 284.59,Z 494.144,A -85,B 0,C 180,E1 -17348.452,E2 -17348.452} C_VEL
LIN {X 0,Y 282.649,Z 504.114,A -85,B 0,C 180,E1 -17350.011,E2 -17350.011} C_VEL
LIN {X 0,Y 280.838,Z 513.206,A -85,B 0,C 180,E1 -17351.775,E2 -17351.775} C_VEL
LIN {X 0,Y 279.474,Z 520.746,A -85,B 0,C 180,E1 -17353.569,E2 -17353.569} C_VEL
LIN {X 0,Y 277.948,Z 528.18,A -85,B 0,C 180,E1 -17355.731,E2 -17355.731} C_VEL
LIN {X 0,Y 276.648,Z 535.049,A -85,B 0,C 180,E1 -17358.277,E2 -17358.277} C_VEL
LIN {X 0,Y 275.963,Z 539.615,A -85,B 0,C 180,E1 -17360.475,E2 -17360.475} C_VEL
LIN {X 0,Y 275.608,Z 543.109,A -85,B 0,C 180,E1 -17362.678,E2 -17362.678} C_VEL
LIN {X 0,Y 275.485,Z 544.956,A -85,B 0,C 180,E1 -17364.238,E2 -17364.238} C_VEL
LIN {X 0,Y 275.411,Z 547.157,A -85,B 0,C 180,E1 -17367.077,E2 -17367.077} C_VEL
LIN {X 0,Y 275.412,Z 547.678,A -85,B 0,C 180,E1 -17368.541,E2 -17368.541} C_VEL
LIN {X 0,Y 275.517,Z 547.785,A -85,B 0,C 180,E1 -17370.003,E2 -17370.003} C_VEL
LIN {X 0,Y 275.438,Z 547.487,A -85,B 0,C 180,E1 -17371.465,E2 -17371.465} C_VEL
LIN {X 0,Y 275.422,Z 546.798,A -85,B 0,C 180,E1 -17372.928,E2 -17372.928} C_VEL
LIN {X 0,Y 275.441,Z 545.682,A -85,B 0,C 180,E1 -17374.393,E2 -17374.393} C_VEL
LIN {X 0,Y 275.492,Z 544.118,A -85,B 0,C 180,E1 -17375.86,E2 -17375.86} C_VEL
LIN {X 0,Y 275.701,Z 540.963,A -85,B 0,C 180,E1 -17378.062,E2 -17378.062} C_VEL
LIN {X 0,Y 276.197,Z 536.736,A -85,B 0,C 180,E1 -17380.263,E2 -17380.263} C_VEL
LIN {X 0,Y 277.088,Z 530.295,A -85,B 0,C 180,E1 -17382.825,E2 -17382.825} C_VEL
LIN {X 0,Y 278.357,Z 523.283,A -85,B 0,C 180,E1 -17385.001,E2 -17385.001} C_VEL
LIN {X 0,Y 279.796,Z 515.172,A -85,B 0,C 180,E1 -17387.012,E2 -17387.012} C_VEL
LIN {X 0,Y 281.305,Z 505.472,A -85,B 0,C 180,E1 -17388.955,E2 -17388.955} C_VEL
LIN {X 0,Y 283.056,Z 495.605,A -85,B 0,C 180,E1 -17390.533,E2 -17390.533} C_VEL
LIN {X 0,Y 283.709,Z 490.458,A -85,B 0,C 180,E1 -17391.243,E2 -17391.243} C_VEL
LIN {X 0,Y 283.132,Z 478.5,A -85,B 0,C 180,E1 -17392.746,E2 -17392.746} C_VEL
LIN {X 0,Y 281.97,Z 466.208,A -85,B 0,C 180,E1 -17394.009,E2 -17394.009} C_VEL
LIN {X 0,Y 280.058,Z 453.459,A -85,B 0,C 180,E1 -17395.073,E2 -17395.073} C_VEL
LIN {X 0,Y 277.4,Z 440.17,A -85,B 0,C 180,E1 -17395.955,E2 -17395.955} C_VEL
LIN {X 0,Y 278.449,Z 433.488,A -85,B 0,C 180,E1 -17400.32,E2 -17400.32} C_VEL
LIN {X 0,Y 279.606,Z 427.193,A -85,B 0,C 180,E1 -17404.523,E2 -17404.523} C_VEL
LIN {X 0,Y 280.149,Z 423.599,A -85,B 0,C 180,E1 -17407.022,E2 -17407.022} C_VEL
LIN {X 0,Y 279.736,Z 419.792,A -85,B 0,C 180,E1 -17409.842,E2 -17409.842} C_VEL
LIN {X 0,Y 279.058,Z 415.651,A -85,B 0,C 180,E1 -17413.083,E2 -17413.083} C_VEL
LIN {X 0,Y 278.131,Z 410.848,A -85,B 0,C 180,E1 -17417.124,E2 -17417.124} C_VEL
LIN {X 0,Y 277.292,Z 405.947,A -85,B 0,C 180,E1 -17421.571,E2 -17421.571} C_VEL
LIN {X 0,Y 277.292,Z 405.946,A -85,B 0,C 180,E1 -17424.342,E2 -17424.342} C_VEL
LIN {X 0,Y 277.251,Z 405.95,A -85,B 0,C 180,E1 -17427.837,E2 -17427.837} C_VEL
LIN {X 0,Y 277.275,Z 405.947,A -85,B 0,C 180,E1 -17431.211,E2 -17431.211} C_VEL
LIN {X 0,Y 277.32,Z 405.943,A -85,B 0,C 180,E1 -17434.48,E2 -17434.48} C_VEL
LIN {X 0,Y 277.293,Z 405.942,A -85,B 0,C 180,E1 -17437.655,E2 -17437.655} C_VEL
LIN {X 0,Y 277.353,Z 405.939,A -85,B 0,C 180,E1 -17440.767,E2 -17440.767} C_VEL
LIN {X 0,Y 277.436,Z 405.927,A -85,B 0,C 180,E1 -17445.326,E2 -17445.326} C_VEL
LIN {X 0,Y 277.469,Z 405.923,A -85,B 0,C 180,E1 -17449.787,E2 -17449.787} C_VEL
LIN {X 0,Y 277.648,Z 405.9,A -85,B 0,C 180,E1 -17452.729,E2 -17452.729} C_VEL
LIN {X 0,Y 277.827,Z 405.876,A -85,B 0,C 180,E1 -17458.55,E2 -17458.55} C_VEL
LIN {X 0,Y 277.827,Z 405.876,A -85,B 0,C 180,E1 -17461.449,E2 -17461.449} C_VEL
LIN {X 0,Y 277.66,Z 405.882,A -85,B 0,C 180,E1 -17467.271,E2 -17467.271} C_VEL
LIN {X 0,Y 277.515,Z 405.914,A -85,B 0,C 180,E1 -17470.211,E2 -17470.211} C_VEL
LIN {X 0,Y 277.436,Z 405.924,A -85,B 0,C 180,E1 -17474.674,E2 -17474.674} C_VEL
LIN {X 0,Y 277.352,Z 405.927,A -85,B 0,C 180,E1 -17479.233,E2 -17479.233} C_VEL
LIN {X 0,Y 277.327,Z 405.937,A -85,B 0,C 180,E1 -17484.169,E2 -17484.169} C_VEL
LIN {X 0,Y 277.331,Z 405.941,A -85,B 0,C 180,E1 -17487.503,E2 -17487.503} C_VEL
LIN {X 0,Y 277.28,Z 405.938,A -85,B 0,C 180,E1 -17490.48,E2 -17490.48} C_VEL
LIN {X 0,Y 277.254,Z 405.942,A -85,B 0,C 180,E1 -17493.895,E2 -17493.895} C_VEL
LIN {X 0,Y 277.272,Z 405.948,A -85,B 0,C 180,E1 -17497.469,E2 -17497.469} C_VEL
LIN {X 0,Y 277.217,Z 405.952,A -85,B 0,C 180,E1 -17501.235,E2 -17501.235} C_VEL
LIN {X 0,Y 277.223,Z 405.948,A -85,B 0,C 180,E1 -17505.222,E2 -17505.222} C_VEL
LIN {X 0,Y 277.229,Z 405.951,A -85,B 0,C 180,E1 -17509.511,E2 -17509.511} C_VEL
LIN {X 0,Y 277.271,Z 405.94,A -85,B 0,C 180,E1 -17512.529,E2 -17512.529} C_VEL
LIN {X 0,Y 277.253,Z 405.948,A -85,B 0,C 180,E1 -17516.103,E2 -17516.103} C_VEL
LIN {X 0,Y 277.267,Z 405.942,A -85,B 0,C 180,E1 -17519.537,E2 -17519.537} C_VEL
LIN {X 0,Y 277.361,Z 405.94,A -85,B 0,C 180,E1 -17522.862,E2 -17522.862} C_VEL
LIN {X 0,Y 277.334,Z 405.936,A -85,B 0,C 180,E1 -17526.077,E2 -17526.077} C_VEL
LIN {X 0,Y 277.35,Z 405.936,A -85,B 0,C 180,E1 -17530.764,E2 -17530.764} C_VEL
LIN {X 0,Y 277.44,Z 405.926,A -85,B 0,C 180,E1 -17534.281,E2 -17534.281} C_VEL
LIN {X 0,Y 277.267,Z 405.949,A -85,B 0,C 180,E1 -17538.298,E2 -17538.298} C_VEL
LIN {X 0,Y 277.117,Z 406.318,A -85,B 0,C 180,E1 -17541.527,E2 -17541.527} C_VEL
LIN {X 0,Y 277.144,Z 408.299,A -85,B 0,C 180,E1 -17544.176,E2 -17544.176} C_VEL
LIN {X 0,Y 276.609,Z 410.754,A -85,B 0,C 180,E1 -17547.235,E2 -17547.235} C_VEL
LIN {X 0,Y 280.851,Z 424.374,A -85,B 0,C 180,E1 -17548.351,E2 -17548.351} C_VEL
LIN {X 0,Y 284.2,Z 436.465,A -85,B 0,C 180,E1 -17549.578,E2 -17549.578} C_VEL
LIN {X 0,Y 286.351,Z 447.907,A -85,B 0,C 180,E1 -17550.926,E2 -17550.926} C_VEL
LIN {X 0,Y 284.926,Z 459.244,A -85,B 0,C 180,E1 -17552.294,E2 -17552.294} C_VEL
LIN {X 0,Y 283.291,Z 469.92,A -85,B 0,C 180,E1 -17553.909,E2 -17553.909} C_VEL
LIN {X 0,Y 281.641,Z 479.512,A -85,B 0,C 180,E1 -17555.726,E2 -17555.726} C_VEL
LIN {X 0,Y 279.94,Z 488.773,A -85,B 0,C 180,E1 -17557.934,E2 -17557.934} C_VEL
LIN {X 0,Y 278.532,Z 496.416,A -85,B 0,C 180,E1 -17560.244,E2 -17560.244} C_VEL
LIN {X 0,Y 277.464,Z 502.09,A -85,B 0,C 180,E1 -17562.43,E2 -17562.43} C_VEL
LIN {X 0,Y 276.567,Z 507.303,A -85,B 0,C 180,E1 -17565.063,E2 -17565.063} C_VEL
LIN {X 0,Y 275.849,Z 511.119,A -85,B 0,C 180,E1 -17567.799,E2 -17567.799} C_VEL
LIN {X 0,Y 275.614,Z 512.579,A -85,B 0,C 180,E1 -17569.356,E2 -17569.356} C_VEL
LIN {X 0,Y 275.421,Z 513.621,A -85,B 0,C 180,E1 -17570.927,E2 -17570.927} C_VEL
LIN {X 0,Y 275.371,Z 514.298,A -85,B 0,C 180,E1 -17573.25,E2 -17573.25} C_VEL
LIN {X 0,Y 275.519,Z 513.948,A -85,B 0,C 180,E1 -17575.695,E2 -17575.695} C_VEL
LIN {X 0,Y 275.761,Z 513.107,A -85,B 0,C 180,E1 -17577.302,E2 -17577.302} C_VEL
LIN {X 0,Y 276.465,Z 510.358,A -85,B 0,C 180,E1 -17580.196,E2 -17580.196} C_VEL
LIN {X 0,Y 277.337,Z 506.544,A -85,B 0,C 180,E1 -17582.748,E2 -17582.748} C_VEL
LIN {X 0,Y 278.215,Z 502.743,A -85,B 0,C 180,E1 -17584.633,E2 -17584.633} C_VEL
LIN {X 0,Y 279.687,Z 496.431,A -85,B 0,C 180,E1 -17587.086,E2 -17587.086} C_VEL
LIN {X 0,Y 281.254,Z 489.357,A -85,B 0,C 180,E1 -17589.229,E2 -17589.229} C_VEL
LIN {X 0,Y 282.934,Z 481.423,A -85,B 0,C 180,E1 -17591.162,E2 -17591.162} C_VEL
LIN {X 0,Y 284.703,Z 472.535,A -85,B 0,C 180,E1 -17592.918,E2 -17592.918} C_VEL
LIN {X 0,Y 286.607,Z 462.199,A -85,B 0,C 180,E1 -17594.549,E2 -17594.549} C_VEL
LIN {X 0,Y 288.202,Z 451.981,A -85,B 0,C 180,E1 -17595.839,E2 -17595.839} C_VEL
LIN {X 0,Y 286.616,Z 442.155,A -85,B 0,C 180,E1 -17597.135,E2 -17597.135} C_VEL
LIN {X 0,Y 283.634,Z 430.983,A -85,B 0,C 180,E1 -17598.485,E2 -17598.485} C_VEL
LIN {X 0,Y 279.357,Z 418.913,A -85,B 0,C 180,E1 -17599.796,E2 -17599.796} C_VEL
LIN {X 0,Y 276.885,Z 412.784,A -85,B 0,C 180,E1 -17600.399,E2 -17600.399} C_VEL
LIN {X 0,Y 276.852,Z 412.382,A -85,B 0,C 180,E1 -17600.607,E2 -17600.607} C_VEL
LIN {X 0,Y 277.089,Z 409.858,A -85,B 0,C 180,E1 -17604.313,E2 -17604.313} C_VEL
LIN {X 0,Y 277.218,Z 407.593,A -85,B 0,C 180,E1 -17607.833,E2 -17607.833} C_VEL
LIN {X 0,Y 277.246,Z 406.527,A -85,B 0,C 180,E1 -17609.537,E2 -17609.537} C_VEL
LIN {X 0,Y 277.229,Z 405.954,A -85,B 0,C 180,E1 -17611.206,E2 -17611.206} C_VEL
LIN {X 0,Y 277.309,Z 405.945,A -85,B 0,C 180,E1 -17614.479,E2 -17614.479} C_VEL
LIN {X 0,Y 277.312,Z 405.943,A -85,B 0,C 180,E1 -17617.657,E2 -17617.657} C_VEL
LIN {X 0,Y 277.36,Z 405.938,A -85,B 0,C 180,E1 -17620.767,E2 -17620.767} C_VEL
LIN {X 0,Y 277.411,Z 405.931,A -85,B 0,C 180,E1 -17625.325,E2 -17625.325} C_VEL
LIN {X 0,Y 277.489,Z 405.916,A -85,B 0,C 180,E1 -17629.788,E2 -17629.788} C_VEL
LIN {X 0,Y 277.636,Z 405.897,A -85,B 0,C 180,E1 -17632.729,E2 -17632.729} C_VEL
LIN {X 0,Y 277.806,Z 405.88,A -85,B 0,C 180,E1 -17638.55,E2 -17638.55} C_VEL
LIN {X 0,Y 277.809,Z 405.881,A -85,B 0,C 180,E1 -17641.45,E2 -17641.45} C_VEL
LIN {X 0,Y 277.634,Z 405.902,A -85,B 0,C 180,E1 -17647.272,E2 -17647.272} C_VEL
LIN {X 0,Y 277.452,Z 405.924,A -85,B 0,C 180,E1 -17650.603,E2 -17650.603} C_VEL
LIN {X 0,Y 276.733,Z 406.015,A -85,B 0,C 180,E1 -17651.814,E2 -17651.814} C_VEL
LIN {X 0,Y 273.879,Z 406.371,A -85,B 0,C 180,E1 -17653.787,E2 -17653.787} C_VEL
LIN {X 0,Y 271.47,Z 406.672,A -85,B 0,C 180,E1 -17655.391,E2 -17655.391} C_VEL
LIN {X 0,Y 270.409,Z 406.804,A -85,B 0,C 180,E1 -17656.633,E2 -17656.633} C_VEL
LIN {X 0,Y 270.306,Z 406.814,A -85,B 0,C 180,E1 -17657.054,E2 -17657.054} C_VEL
LIN {X 0,Y 270.309,Z 406.816,A -85,B 0,C 180,E1 -17660.622,E2 -17660.622} C_VEL
LIN {X 0,Y 270.276,Z 406.823,A -85,B 0,C 180,E1 -17664.586,E2 -17664.586} C_VEL
LIN {X 0,Y 270.254,Z 406.827,A -85,B 0,C 180,E1 -17667.911,E2 -17667.911} C_VEL
LIN {X 0,Y 270.169,Z 406.835,A -85,B 0,C 180,E1 -17671.35,E2 -17671.35} C_VEL
LIN {X 0,Y 270.205,Z 406.871,A -85,B 0,C 180,E1 -17674.216,E2 -17674.216} C_VEL
LIN {X 0,Y 270.584,Z 408.848,A -85,B 0,C 180,E1 -17676.683,E2 -17676.683} C_VEL
LIN {X 0,Y 271.167,Z 412.124,A -85,B 0,C 180,E1 -17680.387,E2 -17680.387} C_VEL
LIN {X 0,Y 271.86,Z 415.934,A -85,B 0,C 180,E1 -17684.267,E2 -17684.267} C_VEL
LIN {X 0,Y 272.651,Z 420.406,A -85,B 0,C 180,E1 -17688.376,E2 -17688.376} C_VEL
LIN {X 0,Y 273.304,Z 424.593,A -85,B 0,C 180,E1 -17691.896,E2 -17691.896} C_VEL
LIN {X 0,Y 272.964,Z 428.15,A -85,B 0,C 180,E1 -17694.602,E2 -17694.602} C_VEL
LIN {X 0,Y 271.676,Z 434.076,A -85,B 0,C 180,E1 -17698.847,E2 -17698.847} C_VEL
LIN {X 0,Y 270.898,Z 438.462,A -85,B 0,C 180,E1 -17701.831,E2 -17701.831} C_VEL
LIN {X 0,Y 271.781,Z 441.825,A -85,B 0,C 180,E1 -17702.081,E2 -17702.081} C_VEL
LIN {X 0,Y 274.778,Z 454.341,A -85,B 0,C 180,E1 -17703.157,E2 -17703.157} C_VEL
LIN {X 0,Y 276.966,Z 467.253,A -85,B 0,C 180,E1 -17704.449,E2 -17704.449} C_VEL
LIN {X 0,Y 277.886,Z 478.306,A -85,B 0,C 180,E1 -17705.714,E2 -17705.714} C_VEL
LIN {X 0,Y 278.063,Z 490.283,A -85,B 0,C 180,E1 -17707.332,E2 -17707.332} C_VEL
LIN {X 0,Y 277.755,Z 495.283,A -85,B 0,C 180,E1 -17708.089,E2 -17708.089} C_VEL
LIN {X 0,Y 275.544,Z 505.947,A -85,B 0,C 180,E1 -17709.863,E2 -17709.863} C_VEL
LIN {X 0,Y 273.714,Z 514.815,A -85,B 0,C 180,E1 -17711.71,E2 -17711.71} C_VEL
LIN {X 0,Y 272.332,Z 521.871,A -85,B 0,C 180,E1 -17713.512,E2 -17713.512} C_VEL
LIN {X 0,Y 270.806,Z 528.993,A -85,B 0,C 180,E1 -17715.73,E2 -17715.73} C_VEL
LIN {X 0,Y 269.643,Z 534.721,A -85,B 0,C 180,E1 -17717.968,E2 -17717.968} C_VEL
LIN {X 0,Y 268.945,Z 539.263,A -85,B 0,C 180,E1 -17720.224,E2 -17720.224} C_VEL
LIN {X 0,Y 268.537,Z 542.734,A -85,B 0,C 180,E1 -17722.484,E2 -17722.484} C_VEL
LIN {X 0,Y 268.379,Z 544.816,A -85,B 0,C 180,E1 -17724.329,E2 -17724.329} C_VEL
LIN {X 0,Y 268.34,Z 546.751,A -85,B 0,C 180,E1 -17727,E2 -17727} C_VEL
LIN {X 0,Y 268.332,Z 547.251,A -85,B 0,C 180,E1 -17728.502,E2 -17728.502} C_VEL
LIN {X 0,Y 268.429,Z 547.347,A -85,B 0,C 180,E1 -17730.003,E2 -17730.003} C_VEL
LIN {X 0,Y 268.356,Z 547.038,A -85,B 0,C 180,E1 -17731.504,E2 -17731.504} C_VEL
LIN {X 0,Y 268.351,Z 546.339,A -85,B 0,C 180,E1 -17733.005,E2 -17733.005} C_VEL
LIN {X 0,Y 268.393,Z 543.996,A -85,B 0,C 180,E1 -17735.701,E2 -17735.701} C_VEL
LIN {X 0,Y 268.633,Z 540.44,A -85,B 0,C 180,E1 -17738.276,E2 -17738.276} C_VEL
LIN {X 0,Y 269.168,Z 536.185,A -85,B 0,C 180,E1 -17740.534,E2 -17740.534} C_VEL
LIN {X 0,Y 270.132,Z 529.717,A -85,B 0,C 180,E1 -17743.161,E2 -17743.161} C_VEL
LIN {X 0,Y 271.426,Z 522.654,A -85,B 0,C 180,E1 -17745.393,E2 -17745.393} C_VEL
LIN {X 0,Y 272.71,Z 516.036,A -85,B 0,C 180,E1 -17747.1,E2 -17747.1} C_VEL
LIN {X 0,Y 274.207,Z 506.716,A -85,B 0,C 180,E1 -17749.076,E2 -17749.076} C_VEL
LIN {X 0,Y 276.171,Z 496.007,A -85,B 0,C 180,E1 -17750.874,E2 -17750.874} C_VEL
LIN {X 0,Y 276.811,Z 490.946,A -85,B 0,C 180,E1 -17751.604,E2 -17751.604} C_VEL
LIN {X 0,Y 276.324,Z 479.177,A -85,B 0,C 180,E1 -17753.156,E2 -17753.156} C_VEL
LIN {X 0,Y 275.244,Z 467.143,A -85,B 0,C 180,E1 -17754.453,E2 -17754.453} C_VEL
LIN {X 0,Y 273.354,Z 454.123,A -85,B 0,C 180,E1 -17755.595,E2 -17755.595} C_VEL
LIN {X 0,Y 270.562,Z 440.632,A -85,B 0,C 180,E1 -17756.523,E2 -17756.523} C_VEL
LIN {X 0,Y 270.486,Z 439.812,A -85,B 0,C 180,E1 -17756.579,E2 -17756.579} C_VEL
LIN {X 0,Y 271.364,Z 434.206,A -85,B 0,C 180,E1 -17760.336,E2 -17760.336} C_VEL
LIN {X 0,Y 272.551,Z 428.062,A -85,B 0,C 180,E1 -17764.564,E2 -17764.564} C_VEL
LIN {X 0,Y 273.119,Z 424.504,A -85,B 0,C 180,E1 -17767.088,E2 -17767.088} C_VEL
LIN {X 0,Y 272.664,Z 420.549,A -85,B 0,C 180,E1 -17770.122,E2 -17770.122} C_VEL
LIN {X 0,Y 271.813,Z 415.441,A -85,B 0,C 180,E1 -17774.279,E2 -17774.279} C_VEL
LIN {X 0,Y 271.046,Z 411.62,A -85,B 0,C 180,E1 -17777.611,E2 -17777.611} C_VEL
LIN {X 0,Y 270.266,Z 407.051,A -85,B 0,C 180,E1 -17781.859,E2 -17781.859} C_VEL
LIN {X 0,Y 270.225,Z 406.825,A -85,B 0,C 180,E1 -17783.26,E2 -17783.26} C_VEL
LIN {X 0,Y 270.211,Z 406.83,A -85,B 0,C 180,E1 -17786.893,E2 -17786.893} C_VEL
LIN {X 0,Y 270.203,Z 406.83,A -85,B 0,C 180,E1 -17790.383,E2 -17790.383} C_VEL
LIN {X 0,Y 270.27,Z 406.817,A -85,B 0,C 180,E1 -17793.764,E2 -17793.764} C_VEL
LIN {X 0,Y 270.241,Z 406.822,A -85,B 0,C 180,E1 -17797.039,E2 -17797.039} C_VEL
LIN {X 0,Y 270.31,Z 406.817,A -85,B 0,C 180,E1 -17800.245,E2 -17800.245} C_VEL
LIN {X 0,Y 270.405,Z 406.804,A -85,B 0,C 180,E1 -17804.935,E2 -17804.935} C_VEL
LIN {X 0,Y 270.421,Z 406.8,A -85,B 0,C 180,E1 -17809.518,E2 -17809.518} C_VEL
LIN {X 0,Y 270.606,Z 406.778,A -85,B 0,C 180,E1 -17812.539,E2 -17812.539} C_VEL
LIN {X 0,Y 270.793,Z 406.753,A -85,B 0,C 180,E1 -17818.513,E2 -17818.513} C_VEL
LIN {X 0,Y 270.793,Z 406.752,A -85,B 0,C 180,E1 -17821.487,E2 -17821.487} C_VEL
LIN {X 0,Y 270.619,Z 406.759,A -85,B 0,C 180,E1 -17827.461,E2 -17827.461} C_VEL
LIN {X 0,Y 270.45,Z 406.792,A -85,B 0,C 180,E1 -17830.481,E2 -17830.481} C_VEL
LIN {X 0,Y 270.404,Z 406.8,A -85,B 0,C 180,E1 -17835.064,E2 -17835.064} C_VEL
LIN {X 0,Y 270.309,Z 406.8,A -85,B 0,C 180,E1 -17839.755,E2 -17839.755} C_VEL
LIN {X 0,Y 270.282,Z 406.814,A -85,B 0,C 180,E1 -17844.585,E2 -17844.585} C_VEL
LIN {X 0,Y 270.278,Z 406.816,A -85,B 0,C 180,E1 -17847.908,E2 -17847.908} C_VEL
LIN {X 0,Y 270.191,Z 406.82,A -85,B 0,C 180,E1 -17851.347,E2 -17851.347} C_VEL
LIN {X 0,Y 270.209,Z 406.819,A -85,B 0,C 180,E1 -17854.904,E2 -17854.904} C_VEL
LIN {X 0,Y 270.205,Z 406.826,A -85,B 0,C 180,E1 -17858.709,E2 -17858.709} C_VEL
LIN {X 0,Y 270.178,Z 406.822,A -85,B 0,C 180,E1 -17863.249,E2 -17863.249} C_VEL
LIN {X 0,Y 270.181,Z 406.83,A -85,B 0,C 180,E1 -17867.441,E2 -17867.441} C_VEL
LIN {X 0,Y 270.214,Z 406.82,A -85,B 0,C 180,E1 -17871.373,E2 -17871.373} C_VEL
LIN {X 0,Y 270.208,Z 406.828,A -85,B 0,C 180,E1 -17875.093,E2 -17875.093} C_VEL
LIN {X 0,Y 270.206,Z 406.824,A -85,B 0,C 180,E1 -17879.129,E2 -17879.129} C_VEL
LIN {X 0,Y 270.27,Z 406.819,A -85,B 0,C 180,E1 -17882.144,E2 -17882.144} C_VEL
LIN {X 0,Y 270.282,Z 406.814,A -85,B 0,C 180,E1 -17885.517,E2 -17885.517} C_VEL
LIN {X 0,Y 270.307,Z 406.814,A -85,B 0,C 180,E1 -17890.242,E2 -17890.242} C_VEL
LIN {X 0,Y 270.393,Z 406.805,A -85,B 0,C 180,E1 -17894.932,E2 -17894.932} C_VEL
LIN {X 0,Y 270.232,Z 406.824,A -85,B 0,C 180,E1 -17897.989,E2 -17897.989} C_VEL
LIN {X 0,Y 270.07,Z 406.961,A -85,B 0,C 180,E1 -17901.015,E2 -17901.015} C_VEL
LIN {X 0,Y 270.108,Z 409.149,A -85,B 0,C 180,E1 -17904.023,E2 -17904.023} C_VEL
LIN {X 0,Y 269.68,Z 411.123,A -85,B 0,C 180,E1 -17906.589,E2 -17906.589} C_VEL
LIN {X 0,Y 273.384,Z 423.05,A -85,B 0,C 180,E1 -17907.582,E2 -17907.582} C_VEL
LIN {X 0,Y 276.952,Z 435.951,A -85,B 0,C 180,E1 -17908.904,E2 -17908.904} C_VEL
LIN {X 0,Y 278.963,Z 445.099,A -85,B 0,C 180,E1 -17909.997,E2 -17909.997} C_VEL
LIN {X 0,Y 279.627,Z 449.292,A -85,B 0,C 180,E1 -17910.537,E2 -17910.537} C_VEL
LIN {X 0,Y 278.073,Z 460.843,A -85,B 0,C 180,E1 -17911.989,E2 -17911.989} C_VEL
LIN {X 0,Y 276.381,Z 471.304,A -85,B 0,C 180,E1 -17913.642,E2 -17913.642} C_VEL
LIN {X 0,Y 274.626,Z 480.953,A -85,B 0,C 180,E1 -17915.561,E2 -17915.561} C_VEL
LIN {X 0,Y 272.918,Z 489.836,A -85,B 0,C 180,E1 -17917.767,E2 -17917.767} C_VEL
LIN {X 0,Y 271.789,Z 495.727,A -85,B 0,C 180,E1 -17919.583,E2 -17919.583} C_VEL
LIN {X 0,Y 270.581,Z 502.048,A -85,B 0,C 180,E1 -17921.99,E2 -17921.99} C_VEL
LIN {X 0,Y 269.727,Z 506.765,A -85,B 0,C 180,E1 -17924.328,E2 -17924.328} C_VEL
LIN {X 0,Y 269.03,Z 510.344,A -85,B 0,C 180,E1 -17926.697,E2 -17926.697} C_VEL
LIN {X 0,Y 268.505,Z 513.207,A -85,B 0,C 180,E1 -17929.561,E2 -17929.561} C_VEL
LIN {X 0,Y 268.301,Z 514.31,A -85,B 0,C 180,E1 -17931.51,E2 -17931.51} C_VEL
LIN {X 0,Y 268.31,Z 514.761,A -85,B 0,C 180,E1 -17933.541,E2 -17933.541} C_VEL
LIN {X 0,Y 268.536,Z 514.125,A -85,B 0,C 180,E1 -17936.414,E2 -17936.414} C_VEL
LIN {X 0,Y 268.816,Z 513.116,A -85,B 0,C 180,E1 -17938.069,E2 -17938.069} C_VEL
LIN {X 0,Y 269.542,Z 510.569,A -85,B 0,C 180,E1 -17940.634,E2 -17940.634} C_VEL
LIN {X 0,Y 270.392,Z 506.95,A -85,B 0,C 180,E1 -17943.077,E2 -17943.077} C_VEL
LIN {X 0,Y 271.647,Z 501.811,A -85,B 0,C 180,E1 -17945.595,E2 -17945.595} C_VEL
LIN {X 0,Y 273.266,Z 495.074,A -85,B 0,C 180,E1 -17948.111,E2 -17948.111} C_VEL
LIN {X 0,Y 274.95,Z 488.15,A -85,B 0,C 180,E1 -17950.144,E2 -17950.144} C_VEL
LIN {X 0,Y 276.807,Z 479.41,A -85,B 0,C 180,E1 -17952.208,E2 -17952.208} C_VEL
LIN {X 0,Y 278.93,Z 469.238,A -85,B 0,C 180,E1 -17954.106,E2 -17954.106} C_VEL
LIN {X 0,Y 280.726,Z 459.053,A -85,B 0,C 180,E1 -17955.632,E2 -17955.632} C_VEL
LIN {X 0,Y 281.679,Z 453.327,A -85,B 0,C 180,E1 -17956.344,E2 -17956.344} C_VEL
LIN {X 0,Y 280.103,Z 443.692,A -85,B 0,C 180,E1 -17957.69,E2 -17957.69} C_VEL
LIN {X 0,Y 277.312,Z 433.075,A -85,B 0,C 180,E1 -17959.045,E2 -17959.045} C_VEL
LIN {X 0,Y 273.076,Z 421.15,A -85,B 0,C 180,E1 -17960.433,E2 -17960.433} C_VEL
LIN {X 0,Y 270.024,Z 413.844,A -85,B 0,C 180,E1 -17961.224,E2 -17961.224} C_VEL
LIN {X 0,Y 269.883,Z 412.98,A -85,B 0,C 180,E1 -17961.319,E2 -17961.319} C_VEL
LIN {X 0,Y 270.104,Z 410.508,A -85,B 0,C 180,E1 -17965.08,E2 -17965.08} C_VEL
LIN {X 0,Y 270.239,Z 407.999,A -85,B 0,C 180,E1 -17969.109,E2 -17969.109} C_VEL
LIN {X 0,Y 270.194,Z 407.261,A -85,B 0,C 180,E1 -17970.382,E2 -17970.382} C_VEL
LIN {X 0,Y 270.245,Z 406.823,A -85,B 0,C 180,E1 -17972.145,E2 -17972.145} C_VEL
LIN {X 0,Y 270.299,Z 406.82,A -85,B 0,C 180,E1 -17975.5,E2 -17975.5} C_VEL
LIN {X 0,Y 270.315,Z 406.813,A -85,B 0,C 180,E1 -17980.246,E2 -17980.246} C_VEL
LIN {X 0,Y 270.379,Z 406.805,A -85,B 0,C 180,E1 -17984.934,E2 -17984.934} C_VEL
LIN {X 0,Y 270.424,Z 406.796,A -85,B 0,C 180,E1 -17989.518,E2 -17989.518} C_VEL
LIN {X 0,Y 270.594,Z 406.775,A -85,B 0,C 180,E1 -17992.538,E2 -17992.538} C_VEL
LIN {X 0,Y 270.771,Z 406.757,A -85,B 0,C 180,E1 -17998.513,E2 -17998.513} C_VEL
LIN {X 0,Y 270.775,Z 406.757,A -85,B 0,C 180,E1 -18001.487,E2 -18001.487} C_VEL
LIN {X 0,Y 270.593,Z 406.779,A -85,B 0,C 180,E1 -18007.462,E2 -18007.462} C_VEL
LIN {X 0,Y 270.416,Z 406.8,A -85,B 0,C 180,E1 -18010.577,E2 -18010.577} C_VEL
LIN {X 0,Y 270.386,Z 406.806,A -85,B 0,C 180,E1 -18015.066,E2 -18015.066} C_VEL
LIN {X 0,Y 270.306,Z 406.814,A -85,B 0,C 180,E1 -18017.054,E2 -18017.054} C_VEL
LIN {X 0,Y 269.597,Z 406.906,A -85,B 0,C 180,E1 -18018.297,E2 -18018.297} C_VEL
LIN {X 0,Y 266.745,Z 407.263,A -85,B 0,C 180,E1 -18020.324,E2 -18020.324} C_VEL
LIN {X 0,Y 264.342,Z 407.565,A -85,B 0,C 180,E1 -18021.972,E2 -18021.972} C_VEL
LIN {X 0,Y 263.3,Z 407.693,A -85,B 0,C 180,E1 -18023.249,E2 -18023.249} C_VEL
LIN {X 0,Y 263.208,Z 407.702,A -85,B 0,C 180,E1 -18023.681,E2 -18023.681} C_VEL
LIN {X 0,Y 263.181,Z 407.708,A -85,B 0,C 180,E1 -18028.217,E2 -18028.217} C_VEL
LIN {X 0,Y 263.157,Z 407.709,A -85,B 0,C 180,E1 -18033.138,E2 -18033.138} C_VEL
LIN {X 0,Y 263.696,Z 410.619,A -85,B 0,C 180,E1 -18036.919,E2 -18036.919} C_VEL
LIN {X 0,Y 264.434,Z 414.794,A -85,B 0,C 180,E1 -18041.639,E2 -18041.639} C_VEL
LIN {X 0,Y 264.928,Z 417.345,A -85,B 0,C 180,E1 -18044.259,E2 -18044.259} C_VEL
LIN {X 0,Y 265.706,Z 421.963,A -85,B 0,C 180,E1 -18048.609,E2 -18048.609} C_VEL
LIN {X 0,Y 266.267,Z 425.415,A -85,B 0,C 180,E1 -18051.603,E2 -18051.603} C_VEL
LIN {X 0,Y 265.95,Z 429.029,A -85,B 0,C 180,E1 -18054.457,E2 -18054.457} C_VEL
LIN {X 0,Y 264.596,Z 435.098,A -85,B 0,C 180,E1 -18058.903,E2 -18058.903} C_VEL
LIN {X 0,Y 264.062,Z 438.07,A -85,B 0,C 180,E1 -18060.935,E2 -18060.935} C_VEL
LIN {X 0,Y 265.766,Z 444.426,A -85,B 0,C 180,E1 -18061.456,E2 -18061.456} C_VEL
LIN {X 0,Y 268.506,Z 455.908,A -85,B 0,C 180,E1 -18062.535,E2 -18062.535} C_VEL
LIN {X 0,Y 270.388,Z 467.692,A -85,B 0,C 180,E1 -18063.781,E2 -18063.781} C_VEL
LIN {X 0,Y 271.27,Z 478.328,A -85,B 0,C 180,E1 -18065.064,E2 -18065.064} C_VEL
LIN {X 0,Y 271.357,Z 490.277,A -85,B 0,C 180,E1 -18066.74,E2 -18066.74} C_VEL
LIN {X 0,Y 270.948,Z 496.411,A -85,B 0,C 180,E1 -18067.71,E2 -18067.71} C_VEL
LIN {X 0,Y 268.884,Z 505.835,A -85,B 0,C 180,E1 -18069.341,E2 -18069.341} C_VEL
LIN {X 0,Y 266.992,Z 514.479,A -85,B 0,C 180,E1 -18071.192,E2 -18071.192} C_VEL
LIN {X 0,Y 265.523,Z 521.657,A -85,B 0,C 180,E1 -18073.076,E2 -18073.076} C_VEL
LIN {X 0,Y 263.901,Z 528.72,A -85,B 0,C 180,E1 -18075.348,E2 -18075.348} C_VEL
LIN {X 0,Y 262.653,Z 534.408,A -85,B 0,C 180,E1 -18077.643,E2 -18077.643} C_VEL
LIN {X 0,Y 261.903,Z 538.917,A -85,B 0,C 180,E1 -18079.958,E2 -18079.958} C_VEL
LIN {X 0,Y 261.457,Z 542.359,A -85,B 0,C 180,E1 -18082.279,E2 -18082.279} C_VEL
LIN {X 0,Y 261.276,Z 544.668,A -85,B 0,C 180,E1 -18084.419,E2 -18084.419} C_VEL
LIN {X 0,Y 261.269,Z 546.343,A -85,B 0,C 180,E1 -18086.919,E2 -18086.919} C_VEL
LIN {X 0,Y 261.255,Z 546.824,A -85,B 0,C 180,E1 -18088.461,E2 -18088.461} C_VEL
LIN {X 0,Y 261.344,Z 546.909,A -85,B 0,C 180,E1 -18090.003,E2 -18090.003} C_VEL
LIN {X 0,Y 261.277,Z 546.59,A -85,B 0,C 180,E1 -18091.544,E2 -18091.544} C_VEL
LIN {X 0,Y 261.283,Z 545.878,A -85,B 0,C 180,E1 -18093.087,E2 -18093.087} C_VEL
LIN {X 0,Y 261.298,Z 543.757,A -85,B 0,C 180,E1 -18095.631,E2 -18095.631} C_VEL
LIN {X 0,Y 261.579,Z 539.917,A -85,B 0,C 180,E1 -18098.501,E2 -18098.501} C_VEL
LIN {X 0,Y 262.132,Z 535.634,A -85,B 0,C 180,E1 -18100.82,E2 -18100.82} C_VEL
LIN {X 0,Y 263.199,Z 529.139,A -85,B 0,C 180,E1 -18103.514,E2 -18103.514} C_VEL
LIN {X 0,Y 264.535,Z 522.024,A -85,B 0,C 180,E1 -18105.805,E2 -18105.805} C_VEL
LIN {X 0,Y 265.987,Z 514.388,A -85,B 0,C 180,E1 -18107.787,E2 -18107.787} C_VEL
LIN {X 0,Y 267.464,Z 505.999,A -85,B 0,C 180,E1 -18109.577,E2 -18109.577} C_VEL
LIN {X 0,Y 269.54,Z 495.237,A -85,B 0,C 180,E1 -18111.412,E2 -18111.412} C_VEL
LIN {X 0,Y 269.926,Z 491.422,A -85,B 0,C 180,E1 -18111.982,E2 -18111.982} C_VEL
LIN {X 0,Y 269.519,Z 479.786,A -85,B 0,C 180,E1 -18113.587,E2 -18113.587} C_VEL
LIN {X 0,Y 268.541,Z 468.237,A -85,B 0,C 180,E1 -18114.894,E2 -18114.894} C_VEL
LIN {X 0,Y 266.755,Z 455.575,A -85,B 0,C 180,E1 -18116.071,E2 -18116.071} C_VEL
LIN {X 0,Y 264.018,Z 441.939,A -85,B 0,C 180,E1 -18117.09,E2 -18117.09} C_VEL
LIN {X 0,Y 263.557,Z 439.331,A -85,B 0,C 180,E1 -18117.282,E2 -18117.282} C_VEL
LIN {X 0,Y 264.67,Z 432.827,A -85,B 0,C 180,E1 -18121.818,E2 -18121.818} C_VEL
LIN {X 0,Y 265.781,Z 427.545,A -85,B 0,C 180,E1 -18125.576,E2 -18125.576} C_VEL
LIN {X 0,Y 266.066,Z 424.852,A -85,B 0,C 180,E1 -18127.586,E2 -18127.586} C_VEL
LIN {X 0,Y 265.692,Z 421.906,A -85,B 0,C 180,E1 -18129.906,E2 -18129.906} C_VEL
LIN {X 0,Y 264.963,Z 417.433,A -85,B 0,C 180,E1 -18133.604,E2 -18133.604} C_VEL
LIN {X 0,Y 264.158,Z 413.276,A -85,B 0,C 180,E1 -18137.279,E2 -18137.279} C_VEL
LIN {X 0,Y 263.519,Z 409.69,A -85,B 0,C 180,E1 -18140.665,E2 -18140.665} C_VEL
LIN {X 0,Y 263.194,Z 407.702,A -85,B 0,C 180,E1 -18142.743,E2 -18142.743} C_VEL
LIN {X 0,Y 263.159,Z 407.705,A -85,B 0,C 180,E1 -18145.886,E2 -18145.886} C_VEL
LIN {X 0,Y 263.149,Z 407.707,A -85,B 0,C 180,E1 -18149.506,E2 -18149.506} C_VEL
LIN {X 0,Y 263.199,Z 407.7,A -85,B 0,C 180,E1 -18153.003,E2 -18153.003} C_VEL
LIN {X 0,Y 263.193,Z 407.702,A -85,B 0,C 180,E1 -18156.388,E2 -18156.388} C_VEL
LIN {X 0,Y 263.272,Z 407.691,A -85,B 0,C 180,E1 -18159.694,E2 -18159.694} C_VEL
LIN {X 0,Y 263.353,Z 407.685,A -85,B 0,C 180,E1 -18164.522,E2 -18164.522} C_VEL
LIN {X 0,Y 263.363,Z 407.68,A -85,B 0,C 180,E1 -18169.234,E2 -18169.234} C_VEL
LIN {X 0,Y 263.566,Z 407.657,A -85,B 0,C 180,E1 -18172.338,E2 -18172.338} C_VEL
LIN {X 0,Y 263.758,Z 407.629,A -85,B 0,C 180,E1 -18178.473,E2 -18178.473} C_VEL
LIN {X 0,Y 263.758,Z 407.629,A -85,B 0,C 180,E1 -18181.527,E2 -18181.527} C_VEL
LIN {X 0,Y 263.581,Z 407.635,A -85,B 0,C 180,E1 -18187.661,E2 -18187.661} C_VEL
LIN {X 0,Y 263.382,Z 407.672,A -85,B 0,C 180,E1 -18190.765,E2 -18190.765} C_VEL
LIN {X 0,Y 263.353,Z 407.68,A -85,B 0,C 180,E1 -18195.478,E2 -18195.478} C_VEL
LIN {X 0,Y 263.272,Z 407.675,A -85,B 0,C 180,E1 -18200.306,E2 -18200.306} C_VEL
LIN {X 0,Y 263.216,Z 407.696,A -85,B 0,C 180,E1 -18205.29,E2 -18205.29} C_VEL
LIN {X 0,Y 263.173,Z 407.7,A -85,B 0,C 180,E1 -18208.73,E2 -18208.73} C_VEL
LIN {X 0,Y 263.14,Z 407.691,A -85,B 0,C 180,E1 -18212.287,E2 -18212.287} C_VEL
LIN {X 0,Y 263.189,Z 407.698,A -85,B 0,C 180,E1 -18216.762,E2 -18216.762} C_VEL
LIN {X 0,Y 263.132,Z 407.702,A -85,B 0,C 180,E1 -18221.592,E2 -18221.592} C_VEL
LIN {X 0,Y 263.135,Z 407.703,A -85,B 0,C 180,E1 -18226.015,E2 -18226.015} C_VEL
LIN {X 0,Y 263.112,Z 407.707,A -85,B 0,C 180,E1 -18230.126,E2 -18230.126} C_VEL
LIN {X 0,Y 263.168,Z 407.699,A -85,B 0,C 180,E1 -18234.016,E2 -18234.016} C_VEL
LIN {X 0,Y 263.139,Z 407.706,A -85,B 0,C 180,E1 -18237.71,E2 -18237.71} C_VEL
LIN {X 0,Y 263.206,Z 407.699,A -85,B 0,C 180,E1 -18241.781,E2 -18241.781} C_VEL
LIN {X 0,Y 263.231,Z 407.694,A -85,B 0,C 180,E1 -18245.198,E2 -18245.198} C_VEL
LIN {X 0,Y 263.269,Z 407.69,A -85,B 0,C 180,E1 -18249.691,E2 -18249.691} C_VEL
LIN {X 0,Y 263.346,Z 407.683,A -85,B 0,C 180,E1 -18254.519,E2 -18254.519} C_VEL
LIN {X 0,Y 263.21,Z 407.698,A -85,B 0,C 180,E1 -18257.663,E2 -18257.663} C_VEL
LIN {X 0,Y 263.04,Z 407.798,A -85,B 0,C 180,E1 -18260.772,E2 -18260.772} C_VEL
LIN {X 0,Y 263.098,Z 410.03,A -85,B 0,C 180,E1 -18263.863,E2 -18263.863} C_VEL
LIN {X 0,Y 262.784,Z 411.574,A -85,B 0,C 180,E1 -18265.923,E2 -18265.923} C_VEL
LIN {X 0,Y 266.39,Z 423.347,A -85,B 0,C 180,E1 -18266.925,E2 -18266.925} C_VEL
LIN {X 0,Y 269.682,Z 435.152,A -85,B 0,C 180,E1 -18268.168,E2 -18268.168} C_VEL
LIN {X 0,Y 271.808,Z 443.98,A -85,B 0,C 180,E1 -18269.244,E2 -18269.244} C_VEL
LIN {X 0,Y 272.866,Z 451.05,A -85,B 0,C 180,E1 -18270.182,E2 -18270.182} C_VEL
LIN {X 0,Y 271.206,Z 462.394,A -85,B 0,C 180,E1 -18271.668,E2 -18271.668} C_VEL
LIN {X 0,Y 269.439,Z 472.603,A -85,B 0,C 180,E1 -18273.362,E2 -18273.362} C_VEL
LIN {X 0,Y 267.628,Z 482.193,A -85,B 0,C 180,E1 -18275.348,E2 -18275.348} C_VEL
LIN {X 0,Y 265.909,Z 490.85,A -85,B 0,C 180,E1 -18277.591,E2 -18277.591} C_VEL
LIN {X 0,Y 264.583,Z 497.408,A -85,B 0,C 180,E1 -18279.724,E2 -18279.724} C_VEL
LIN {X 0,Y 263.337,Z 503.694,A -85,B 0,C 180,E1 -18282.325,E2 -18282.325} C_VEL
LIN {X 0,Y 262.524,Z 507.96,A -85,B 0,C 180,E1 -18284.62,E2 -18284.62} C_VEL
LIN {X 0,Y 261.807,Z 511.47,A -85,B 0,C 180,E1 -18287.171,E2 -18287.171} C_VEL
LIN {X 0,Y 261.371,Z 513.818,A -85,B 0,C 180,E1 -18289.76,E2 -18289.76} C_VEL
LIN {X 0,Y 261.188,Z 514.946,A -85,B 0,C 180,E1 -18292.126,E2 -18292.126} C_VEL
LIN {X 0,Y 261.238,Z 515.192,A -85,B 0,C 180,E1 -18293.838,E2 -18293.838} C_VEL
LIN {X 0,Y 261.323,Z 514.953,A -85,B 0,C 180,E1 -18295.483,E2 -18295.483} C_VEL
LIN {X 0,Y 261.64,Z 514.033,A -85,B 0,C 180,E1 -18297.573,E2 -18297.573} C_VEL
LIN {X 0,Y 262.439,Z 511.364,A -85,B 0,C 180,E1 -18300.581,E2 -18300.581} C_VEL
LIN {X 0,Y 263.336,Z 507.781,A -85,B 0,C 180,E1 -18303.165,E2 -18303.165} C_VEL
LIN {X 0,Y 264.643,Z 502.812,A -85,B 0,C 180,E1 -18305.745,E2 -18305.745} C_VEL
LIN {X 0,Y 266.312,Z 496.214,A -85,B 0,C 180,E1 -18308.323,E2 -18308.323} C_VEL
LIN {X 0,Y 268.148,Z 489.013,A -85,B 0,C 180,E1 -18310.529,E2 -18310.529} C_VEL
LIN {X 0,Y 270.045,Z 480.708,A -85,B 0,C 180,E1 -18312.578,E2 -18312.578} C_VEL
LIN {X 0,Y 272.134,Z 471.071,A -85,B 0,C 180,E1 -18314.463,E2 -18314.463} C_VEL
LIN {X 0,Y 274.29,Z 459.73,A -85,B 0,C 180,E1 -18316.227,E2 -18316.227} C_VEL
LIN {X 0,Y 275.134,Z 454.213,A -85,B 0,C 180,E1 -18316.948,E2 -18316.948} C_VEL
LIN {X 0,Y 273.202,Z 443.427,A -85,B 0,C 180,E1 -18318.516,E2 -18318.516} C_VEL
LIN {X 0,Y 269.838,Z 431.401,A -85,B 0,C 180,E1 -18320.106,E2 -18320.106} C_VEL
LIN {X 0,Y 265.531,Z 420.01,A -85,B 0,C 180,E1 -18321.498,E2 -18321.498} C_VEL
LIN {X 0,Y 263.015,Z 414.097,A -85,B 0,C 180,E1 -18322.164,E2 -18322.164} C_VEL
LIN {X 0,Y 262.905,Z 413.486,A -85,B 0,C 180,E1 -18322.231,E2 -18322.231} C_VEL
LIN {X 0,Y 263.136,Z 411.168,A -85,B 0,C 180,E1 -18325.883,E2 -18325.883} C_VEL
LIN {X 0,Y 263.239,Z 409.008,A -85,B 0,C 180,E1 -18329.518,E2 -18329.518} C_VEL
LIN {X 0,Y 263.164,Z 407.727,A -85,B 0,C 180,E1 -18331.79,E2 -18331.79} C_VEL
LIN {X 0,Y 263.223,Z 407.701,A -85,B 0,C 180,E1 -18335.193,E2 -18335.193} C_VEL
LIN {X 0,Y 263.277,Z 407.689,A -85,B 0,C 180,E1 -18339.695,E2 -18339.695} C_VEL
LIN {X 0,Y 263.328,Z 407.681,A -85,B 0,C 180,E1 -18344.521,E2 -18344.521} C_VEL
LIN {X 0,Y 263.357,Z 407.678,A -85,B 0,C 180,E1 -18349.234,E2 -18349.234} C_VEL
LIN {X 0,Y 263.555,Z 407.653,A -85,B 0,C 180,E1 -18352.338,E2 -18352.338} C_VEL
LIN {X 0,Y 263.735,Z 407.633,A -85,B 0,C 180,E1 -18358.473,E2 -18358.473} C_VEL
LIN {X 0,Y 263.74,Z 407.634,A -85,B 0,C 180,E1 -18361.527,E2 -18361.527} C_VEL
LIN {X 0,Y 263.554,Z 407.656,A -85,B 0,C 180,E1 -18367.662,E2 -18367.662} C_VEL
LIN {X 0,Y 263.357,Z 407.679,A -85,B 0,C 180,E1 -18370.766,E2 -18370.766} C_VEL
LIN {X 0,Y 263.334,Z 407.684,A -85,B 0,C 180,E1 -18375.479,E2 -18375.479} C_VEL
LIN {X 0,Y 263.277,Z 407.692,A -85,B 0,C 180,E1 -18380.306,E2 -18380.306} C_VEL
LIN {X 0,Y 263.208,Z 407.702,A -85,B 0,C 180,E1 -18383.681,E2 -18383.681} C_VEL
LIN {X 0,Y 262.511,Z 407.791,A -85,B 0,C 180,E1 -18384.959,E2 -18384.959} C_VEL
LIN {X 0,Y 259.621,Z 408.152,A -85,B 0,C 180,E1 -18387.04,E2 -18387.04} C_VEL
LIN {X 0,Y 257.181,Z 408.454,A -85,B 0,C 180,E1 -18388.733,E2 -18388.733} C_VEL
LIN {X 0,Y 256.136,Z 408.584,A -85,B 0,C 180,E1 -18390.046,E2 -18390.046} C_VEL
LIN {X 0,Y 256.051,Z 408.591,A -85,B 0,C 180,E1 -18390.491,E2 -18390.491} C_VEL
LIN {X 0,Y 256.112,Z 408.708,A -85,B 0,C 180,E1 -18392.203,E2 -18392.203} C_VEL
LIN {X 0,Y 256.507,Z 410.839,A -85,B 0,C 180,E1 -18395.126,E2 -18395.126} C_VEL
LIN {X 0,Y 257.029,Z 413.919,A -85,B 0,C 180,E1 -18398.969,E2 -18398.969} C_VEL
LIN {X 0,Y 257.741,Z 417.503,A -85,B 0,C 180,E1 -18402.976,E2 -18402.976} C_VEL
LIN {X 0,Y 258.479,Z 421.778,A -85,B 0,C 180,E1 -18407.234,E2 -18407.234} C_VEL
LIN {X 0,Y 259.24,Z 426.405,A -85,B 0,C 180,E1 -18411.43,E2 -18411.43} C_VEL
LIN {X 0,Y 259.168,Z 428.768,A -85,B 0,C 180,E1 -18413.379,E2 -18413.379} C_VEL
LIN {X 0,Y 258.099,Z 433.463,A -85,B 0,C 180,E1 -18417.007,E2 -18417.007} C_VEL
LIN {X 0,Y 257.261,Z 437.428,A -85,B 0,C 180,E1 -18419.958,E2 -18419.958} C_VEL
LIN {X 0,Y 258.106,Z 440.779,A -85,B 0,C 180,E1 -18420.232,E2 -18420.232} C_VEL
LIN {X 0,Y 261.43,Z 453.66,A -85,B 0,C 180,E1 -18421.49,E2 -18421.49} C_VEL
LIN {X 0,Y 263.599,Z 466.371,A -85,B 0,C 180,E1 -18422.874,E2 -18422.874} C_VEL
LIN {X 0,Y 264.682,Z 477.826,A -85,B 0,C 180,E1 -18424.304,E2 -18424.304} C_VEL
LIN {X 0,Y 264.727,Z 489.081,A -85,B 0,C 180,E1 -18425.92,E2 -18425.92} C_VEL
LIN {X 0,Y 264.373,Z 496.394,A -85,B 0,C 180,E1 -18427.125,E2 -18427.125} C_VEL
LIN {X 0,Y 262.25,Z 505.731,A -85,B 0,C 180,E1 -18428.794,E2 -18428.794} C_VEL
LIN {X 0,Y 260.246,Z 514.297,A -85,B 0,C 180,E1 -18430.685,E2 -18430.685} C_VEL
LIN {X 0,Y 258.379,Z 522.683,A -85,B 0,C 180,E1 -18433.002,E2 -18433.002} C_VEL
LIN {X 0,Y 256.76,Z 529.474,A -85,B 0,C 180,E1 -18435.337,E2 -18435.337} C_VEL
LIN {X 0,Y 255.402,Z 535.748,A -85,B 0,C 180,E1 -18438.093,E2 -18438.093} C_VEL
LIN {X 0,Y 254.672,Z 539.857,A -85,B 0,C 180,E1 -18440.472,E2 -18440.472} C_VEL
LIN {X 0,Y 254.389,Z 541.996,A -85,B 0,C 180,E1 -18442.063,E2 -18442.063} C_VEL
LIN {X 0,Y 254.174,Z 544.478,A -85,B 0,C 180,E1 -18444.513,E2 -18444.513} C_VEL
LIN {X 0,Y 254.177,Z 545.934,A -85,B 0,C 180,E1 -18446.833,E2 -18446.833} C_VEL
LIN {X 0,Y 254.179,Z 546.398,A -85,B 0,C 180,E1 -18448.419,E2 -18448.419} C_VEL
LIN {X 0,Y 254.261,Z 546.47,A -85,B 0,C 180,E1 -18450.003,E2 -18450.003} C_VEL
LIN {X 0,Y 254.2,Z 546.14,A -85,B 0,C 180,E1 -18451.587,E2 -18451.587} C_VEL
LIN {X 0,Y 254.214,Z 545.412,A -85,B 0,C 180,E1 -18453.173,E2 -18453.173} C_VEL
LIN {X 0,Y 254.208,Z 543.485,A -85,B 0,C 180,E1 -18455.566,E2 -18455.566} C_VEL
LIN {X 0,Y 254.399,Z 540.595,A -85,B 0,C 180,E1 -18457.943,E2 -18457.943} C_VEL
LIN {X 0,Y 254.897,Z 536.651,A -85,B 0,C 180,E1 -18460.327,E2 -18460.327} C_VEL
LIN {X 0,Y 255.858,Z 530.575,A -85,B 0,C 180,E1 -18463.101,E2 -18463.101} C_VEL
LIN {X 0,Y 257.2,Z 523.918,A -85,B 0,C 180,E1 -18465.454,E2 -18465.454} C_VEL
LIN {X 0,Y 258.816,Z 515.837,A -85,B 0,C 180,E1 -18467.738,E2 -18467.738} C_VEL
LIN {X 0,Y 260.37,Z 507.17,A -85,B 0,C 180,E1 -18469.722,E2 -18469.722} C_VEL
LIN {X 0,Y 262.202,Z 497.916,A -85,B 0,C 180,E1 -18471.423,E2 -18471.423} C_VEL
LIN {X 0,Y 263.064,Z 491.825,A -85,B 0,C 180,E1 -18472.38,E2 -18472.38} C_VEL
LIN {X 0,Y 262.702,Z 480.343,A -85,B 0,C 180,E1 -18474.033,E2 -18474.033} C_VEL
LIN {X 0,Y 261.756,Z 468.469,A -85,B 0,C 180,E1 -18475.444,E2 -18475.444} C_VEL
LIN {X 0,Y 259.907,Z 455.57,A -85,B 0,C 180,E1 -18476.7,E2 -18476.7} C_VEL
LIN {X 0,Y 257.289,Z 442.25,A -85,B 0,C 180,E1 -18477.739,E2 -18477.739} C_VEL
LIN {X 0,Y 256.646,Z 438.962,A -85,B 0,C 180,E1 -18477.971,E2 -18477.971} C_VEL
LIN {X 0,Y 257.725,Z 432.951,A -85,B 0,C 180,E1 -18482.29,E2 -18482.29} C_VEL
LIN {X 0,Y 258.664,Z 428.712,A -85,B 0,C 180,E1 -18485.401,E2 -18485.401} C_VEL
LIN {X 0,Y 259.004,Z 425.176,A -85,B 0,C 180,E1 -18488.102,E2 -18488.102} C_VEL
LIN {X 0,Y 258.355,Z 420.836,A -85,B 0,C 180,E1 -18491.695,E2 -18491.695} C_VEL
LIN {X 0,Y 257.604,Z 416.857,A -85,B 0,C 180,E1 -18495.184,E2 -18495.184} C_VEL
LIN {X 0,Y 256.881,Z 412.808,A -85,B 0,C 180,E1 -18498.958,E2 -18498.958} C_VEL
LIN {X 0,Y 256.144,Z 408.579,A -85,B 0,C 180,E1 -18503.361,E2 -18503.361} C_VEL
LIN {X 0,Y 256.076,Z 408.591,A -85,B 0,C 180,E1 -18506.708,E2 -18506.708} C_VEL
LIN {X 0,Y 256.112,Z 408.587,A -85,B 0,C 180,E1 -18510.4,E2 -18510.4} C_VEL
LIN {X 0,Y 256.197,Z 408.573,A -85,B 0,C 180,E1 -18514.863,E2 -18514.863} C_VEL
LIN {X 0,Y 256.176,Z 408.576,A -85,B 0,C 180,E1 -18519.105,E2 -18519.105} C_VEL
LIN {X 0,Y 256.303,Z 408.562,A -85,B 0,C 180,E1 -18524.085,E2 -18524.085} C_VEL
LIN {X 0,Y 256.302,Z 408.56,A -85,B 0,C 180,E1 -18527.328,E2 -18527.328} C_VEL
LIN {X 0,Y 256.524,Z 408.534,A -85,B 0,C 180,E1 -18532.126,E2 -18532.126} C_VEL
LIN {X 0,Y 256.504,Z 408.532,A -85,B 0,C 180,E1 -18536.859,E2 -18536.859} C_VEL
LIN {X 0,Y 256.765,Z 408.502,A -85,B 0,C 180,E1 -18540,E2 -18540} C_VEL
LIN {X 0,Y 256.504,Z 408.529,A -85,B 0,C 180,E1 -18543.141,E2 -18543.141} C_VEL
LIN {X 0,Y 256.548,Z 408.511,A -85,B 0,C 180,E1 -18547.873,E2 -18547.873} C_VEL
LIN {X 0,Y 256.318,Z 408.552,A -85,B 0,C 180,E1 -18551.066,E2 -18551.066} C_VEL
LIN {X 0,Y 256.303,Z 408.556,A -85,B 0,C 180,E1 -18555.915,E2 -18555.915} C_VEL
LIN {X 0,Y 256.175,Z 408.557,A -85,B 0,C 180,E1 -18560.894,E2 -18560.894} C_VEL
LIN {X 0,Y 256.196,Z 408.57,A -85,B 0,C 180,E1 -18565.137,E2 -18565.137} C_VEL
LIN {X 0,Y 256.111,Z 408.578,A -85,B 0,C 180,E1 -18569.6,E2 -18569.6} C_VEL
LIN {X 0,Y 256.075,Z 408.572,A -85,B 0,C 180,E1 -18573.292,E2 -18573.292} C_VEL
LIN {X 0,Y 256.122,Z 408.581,A -85,B 0,C 180,E1 -18577.269,E2 -18577.269} C_VEL
LIN {X 0,Y 256.062,Z 408.585,A -85,B 0,C 180,E1 -18581.202,E2 -18581.202} C_VEL
LIN {X 0,Y 256.069,Z 408.584,A -85,B 0,C 180,E1 -18585.528,E2 -18585.528} C_VEL
LIN {X 0,Y 256.062,Z 408.589,A -85,B 0,C 180,E1 -18588.795,E2 -18588.795} C_VEL
LIN {X 0,Y 256.136,Z 408.572,A -85,B 0,C 180,E1 -18592.866,E2 -18592.866} C_VEL
LIN {X 0,Y 256.074,Z 408.59,A -85,B 0,C 180,E1 -18596.705,E2 -18596.705} C_VEL
LIN {X 0,Y 256.119,Z 408.576,A -85,B 0,C 180,E1 -18600.398,E2 -18600.398} C_VEL
LIN {X 0,Y 256.194,Z 408.573,A -85,B 0,C 180,E1 -18604.859,E2 -18604.859} C_VEL
LIN {X 0,Y 256.172,Z 408.576,A -85,B 0,C 180,E1 -18609.103,E2 -18609.103} C_VEL
LIN {X 0,Y 256.298,Z 408.558,A -85,B 0,C 180,E1 -18614.082,E2 -18614.082} C_VEL
LIN {X 0,Y 256.178,Z 408.574,A -85,B 0,C 180,E1 -18617.319,E2 -18617.319} C_VEL
LIN {X 0,Y 256.006,Z 408.636,A -85,B 0,C 180,E1 -18620.516,E2 -18620.516} C_VEL
LIN {X 0,Y 256.065,Z 410.861,A -85,B 0,C 180,E1 -18623.694,E2 -18623.694} C_VEL
LIN {X 0,Y 255.897,Z 412.067,A -85,B 0,C 180,E1 -18625.222,E2 -18625.222} C_VEL
LIN {X 0,Y 259.678,Z 424.529,A -85,B 0,C 180,E1 -18626.332,E2 -18626.332} C_VEL
LIN {X 0,Y 262.858,Z 435.965,A -85,B 0,C 180,E1 -18627.584,E2 -18627.584} C_VEL
LIN {X 0,Y 265.212,Z 445.905,A -85,B 0,C 180,E1 -18628.858,E2 -18628.858} C_VEL
LIN {X 0,Y 266.141,Z 451.338,A -85,B 0,C 180,E1 -18629.619,E2 -18629.619} C_VEL
LIN {X 0,Y 264.564,Z 462.625,A -85,B 0,C 180,E1 -18631.139,E2 -18631.139} C_VEL
LIN {X 0,Y 262.714,Z 472.882,A -85,B 0,C 180,E1 -18632.872,E2 -18632.872} C_VEL
LIN {X 0,Y 260.789,Z 482.814,A -85,B 0,C 180,E1 -18634.982,E2 -18634.982} C_VEL
LIN {X 0,Y 259.191,Z 490.488,A -85,B 0,C 180,E1 -18637.005,E2 -18637.005} C_VEL
LIN {X 0,Y 257.633,Z 497.822,A -85,B 0,C 180,E1 -18639.417,E2 -18639.417} C_VEL
LIN {X 0,Y 256.45,Z 503.635,A -85,B 0,C 180,E1 -18641.858,E2 -18641.858} C_VEL
LIN {X 0,Y 255.541,Z 508.195,A -85,B 0,C 180,E1 -18644.328,E2 -18644.328} C_VEL
LIN {X 0,Y 255.044,Z 510.617,A -85,B 0,C 180,E1 -18645.992,E2 -18645.992} C_VEL
LIN {X 0,Y 254.622,Z 512.538,A -85,B 0,C 180,E1 -18647.672,E2 -18647.672} C_VEL
LIN {X 0,Y 254.271,Z 514.424,A -85,B 0,C 180,E1 -18649.99,E2 -18649.99} C_VEL
LIN {X 0,Y 254.115,Z 515.517,A -85,B 0,C 180,E1 -18652.776,E2 -18652.776} C_VEL
LIN {X 0,Y 254.176,Z 515.587,A -85,B 0,C 180,E1 -18654.5,E2 -18654.5} C_VEL
LIN {X 0,Y 254.321,Z 515.22,A -85,B 0,C 180,E1 -18656.237,E2 -18656.237} C_VEL
LIN {X 0,Y 254.654,Z 514.324,A -85,B 0,C 180,E1 -18657.976,E2 -18657.976} C_VEL
LIN {X 0,Y 255.082,Z 512.958,A -85,B 0,C 180,E1 -18659.727,E2 -18659.727} C_VEL
LIN {X 0,Y 255.949,Z 509.925,A -85,B 0,C 180,E1 -18662.369,E2 -18662.369} C_VEL
LIN {X 0,Y 257.149,Z 505.567,A -85,B 0,C 180,E1 -18665.021,E2 -18665.021} C_VEL
LIN {X 0,Y 258.668,Z 500.244,A -85,B 0,C 180,E1 -18667.445,E2 -18667.445} C_VEL
LIN {X 0,Y 260.399,Z 493.488,A -85,B 0,C 180,E1 -18669.861,E2 -18669.861} C_VEL
LIN {X 0,Y 262.367,Z 485.816,A -85,B 0,C 180,E1 -18672.037,E2 -18672.037} C_VEL
LIN {X 0,Y 264.571,Z 476.348,A -85,B 0,C 180,E1 -18674.175,E2 -18674.175} C_VEL
LIN {X 0,Y 266.929,Z 465.385,A -85,B 0,C 180,E1 -18676.112,E2 -18676.112} C_VEL
LIN {X 0,Y 268.609,Z 456.379,A -85,B 0,C 180,E1 -18677.386,E2 -18677.386} C_VEL
LIN {X 0,Y 267.129,Z 446.758,A -85,B 0,C 180,E1 -18678.873,E2 -18678.873} C_VEL
LIN {X 0,Y 264.282,Z 435.69,A -85,B 0,C 180,E1 -18680.455,E2 -18680.455} C_VEL
LIN {X 0,Y 260.086,Z 423.912,A -85,B 0,C 180,E1 -18682.005,E2 -18682.005} C_VEL
LIN {X 0,Y 256.182,Z 414.941,A -85,B 0,C 180,E1 -18683.122,E2 -18683.122} C_VEL
LIN {X 0,Y 255.996,Z 413.99,A -85,B 0,C 180,E1 -18683.214,E2 -18683.214} C_VEL
LIN {X 0,Y 256.127,Z 411.871,A -85,B 0,C 180,E1 -18686.716,E2 -18686.716} C_VEL
LIN {X 0,Y 256.232,Z 410.768,A -85,B 0,C 180,E1 -18688.592,E2 -18688.592} C_VEL
LIN {X 0,Y 256.139,Z 408.798,A -85,B 0,C 180,E1 -18692.196,E2 -18692.196} C_VEL
LIN {X 0,Y 256.174,Z 408.578,A -85,B 0,C 180,E1 -18695.7,E2 -18695.7} C_VEL
LIN {X 0,Y 256.227,Z 408.569,A -85,B 0,C 180,E1 -18699.11,E2 -18699.11} C_VEL
LIN {X 0,Y 256.278,Z 408.559,A -85,B 0,C 180,E1 -18704.084,E2 -18704.084} C_VEL
LIN {X 0,Y 256.292,Z 408.56,A -85,B 0,C 180,E1 -18708.933,E2 -18708.933} C_VEL
LIN {X 0,Y 256.523,Z 408.53,A -85,B 0,C 180,E1 -18712.127,E2 -18712.127} C_VEL
LIN {X 0,Y 256.698,Z 408.51,A -85,B 0,C 180,E1 -18718.431,E2 -18718.431} C_VEL
LIN {X 0,Y 256.705,Z 408.51,A -85,B 0,C 180,E1 -18721.569,E2 -18721.569} C_VEL
LIN {X 0,Y 256.522,Z 408.532,A -85,B 0,C 180,E1 -18727.874,E2 -18727.874} C_VEL
LIN {X 0,Y 256.293,Z 408.559,A -85,B 0,C 180,E1 -18731.067,E2 -18731.067} C_VEL
LIN {X 0,Y 256.283,Z 408.562,A -85,B 0,C 180,E1 -18735.916,E2 -18735.916} C_VEL
LIN {X 0,Y 256.228,Z 408.571,A -85,B 0,C 180,E1 -18740.89,E2 -18740.89} C_VEL
LIN {X 0,Y 256.182,Z 408.579,A -85,B 0,C 180,E1 -18745.145,E2 -18745.145} C_VEL
LIN {X 0,Y 256.089,Z 408.591,A -85,B 0,C 180,E1 -18749.603,E2 -18749.603} C_VEL
LIN {X 0,Y 256.051,Z 408.591,A -85,B 0,C 180,E1 -18750.491,E2 -18750.491} C_VEL
LIN {X 0,Y 255.757,Z 408.771,A -85,B 0,C 180,E1 -18751.369,E2 -18751.369} C_VEL
LIN {X 0,Y 254.525,Z 409.567,A -85,B 0,C 180,E1 -18752.659,E2 -18752.659} C_VEL
LIN {X 0,Y 250.689,Z 412.575,A -85,B 0,C 180,E1 -18755.639,E2 -18755.639} C_VEL
LIN {X 0,Y 249.875,Z 413.83,A -85,B 0,C 180,E1 -18756.966,E2 -18756.966} C_VEL
LIN {X 0,Y 249.863,Z 414.188,A -85,B 0,C 180,E1 -18757.416,E2 -18757.416} C_VEL
LIN {X 0,Y 250.394,Z 416.93,A -85,B 0,C 180,E1 -18760.733,E2 -18760.733} C_VEL
LIN {X 0,Y 251.004,Z 420.316,A -85,B 0,C 180,E1 -18764.426,E2 -18764.426} C_VEL
LIN {X 0,Y 251.62,Z 423.782,A -85,B 0,C 180,E1 -18767.912,E2 -18767.912} C_VEL
LIN {X 0,Y 252.242,Z 427.407,A -85,B 0,C 180,E1 -18771.274,E2 -18771.274} C_VEL
LIN {X 0,Y 251.971,Z 430.623,A -85,B 0,C 180,E1 -18773.986,E2 -18773.986} C_VEL
LIN {X 0,Y 250.791,Z 435.521,A -85,B 0,C 180,E1 -18777.834,E2 -18777.834} C_VEL
LIN {X 0,Y 250.46,Z 436.94,A -85,B 0,C 180,E1 -18778.925,E2 -18778.925} C_VEL
LIN {X 0,Y 251.364,Z 440.368,A -85,B 0,C 180,E1 -18779.227,E2 -18779.227} C_VEL
LIN {X 0,Y 254.92,Z 453.857,A -85,B 0,C 180,E1 -18780.627,E2 -18780.627} C_VEL
LIN {X 0,Y 256.888,Z 465.12,A -85,B 0,C 180,E1 -18781.92,E2 -18781.92} C_VEL
LIN {X 0,Y 258.095,Z 477.54,A -85,B 0,C 180,E1 -18783.53,E2 -18783.53} C_VEL
LIN {X 0,Y 258.127,Z 489.404,A -85,B 0,C 180,E1 -18785.305,E2 -18785.305} C_VEL
LIN {X 0,Y 257.6,Z 497.536,A -85,B 0,C 180,E1 -18786.701,E2 -18786.701} C_VEL
LIN {X 0,Y 255.166,Z 507.463,A -85,B 0,C 180,E1 -18788.6,E2 -18788.6} C_VEL
LIN {X 0,Y 252.806,Z 517.163,A -85,B 0,C 180,E1 -18790.945,E2 -18790.945} C_VEL
LIN {X 0,Y 251.235,Z 523.714,A -85,B 0,C 180,E1 -18792.922,E2 -18792.922} C_VEL
LIN {X 0,Y 249.613,Z 530.225,A -85,B 0,C 180,E1 -18795.325,E2 -18795.325} C_VEL
LIN {X 0,Y 248.404,Z 535.433,A -85,B 0,C 180,E1 -18797.752,E2 -18797.752} C_VEL
LIN {X 0,Y 247.637,Z 539.515,A -85,B 0,C 180,E1 -18800.199,E2 -18800.199} C_VEL
LIN {X 0,Y 247.342,Z 541.635,A -85,B 0,C 180,E1 -18801.836,E2 -18801.836} C_VEL
LIN {X 0,Y 247.088,Z 544.25,A -85,B 0,C 180,E1 -18804.576,E2 -18804.576} C_VEL
LIN {X 0,Y 247.087,Z 545.522,A -85,B 0,C 180,E1 -18806.742,E2 -18806.742} C_VEL
LIN {X 0,Y 247.105,Z 545.972,A -85,B 0,C 180,E1 -18808.373,E2 -18808.373} C_VEL
LIN {X 0,Y 247.181,Z 546.031,A -85,B 0,C 180,E1 -18810.003,E2 -18810.003} C_VEL
LIN {X 0,Y 247.126,Z 545.688,A -85,B 0,C 180,E1 -18811.633,E2 -18811.633} C_VEL
LIN {X 0,Y 247.124,Z 544.936,A -85,B 0,C 180,E1 -18813.264,E2 -18813.264} C_VEL
LIN {X 0,Y 247.132,Z 543.165,A -85,B 0,C 180,E1 -18815.53,E2 -18815.53} C_VEL
LIN {X 0,Y 247.355,Z 540.07,A -85,B 0,C 180,E1 -18818.17,E2 -18818.17} C_VEL
LIN {X 0,Y 247.868,Z 536.093,A -85,B 0,C 180,E1 -18820.623,E2 -18820.623} C_VEL
LIN {X 0,Y 248.892,Z 529.964,A -85,B 0,C 180,E1 -18823.474,E2 -18823.474} C_VEL
LIN {X 0,Y 250.274,Z 523.264,A -85,B 0,C 180,E1 -18825.893,E2 -18825.893} C_VEL
LIN {X 0,Y 251.754,Z 516.451,A -85,B 0,C 180,E1 -18827.886,E2 -18827.886} C_VEL
LIN {X 0,Y 253.286,Z 508.22,A -85,B 0,C 180,E1 -18829.874,E2 -18829.874} C_VEL
LIN {X 0,Y 255.338,Z 498.219,A -85,B 0,C 180,E1 -18831.816,E2 -18831.816} C_VEL
LIN {X 0,Y 256.206,Z 493.533,A -85,B 0,C 180,E1 -18832.587,E2 -18832.587} C_VEL
LIN {X 0,Y 255.959,Z 482.186,A -85,B 0,C 180,E1 -18834.325,E2 -18834.325} C_VEL
LIN {X 0,Y 255.198,Z 471.014,A -85,B 0,C 180,E1 -18835.751,E2 -18835.751} C_VEL
LIN {X 0,Y 253.605,Z 458.465,A -85,B 0,C 180,E1 -18837.082,E2 -18837.082} C_VEL
LIN {X 0,Y 251.176,Z 445.537,A -85,B 0,C 180,E1 -18838.199,E2 -18838.199} C_VEL
LIN {X 0,Y 249.718,Z 438.537,A -85,B 0,C 180,E1 -18838.717,E2 -18838.717} C_VEL
LIN {X 0,Y 250.773,Z 433.074,A -85,B 0,C 180,E1 -18842.779,E2 -18842.779} C_VEL
LIN {X 0,Y 251.72,Z 428.899,A -85,B 0,C 180,E1 -18845.935,E2 -18845.935} C_VEL
LIN {X 0,Y 251.906,Z 425.534,A -85,B 0,C 180,E1 -18848.631,E2 -18848.631} C_VEL
LIN {X 0,Y 251.033,Z 420.146,A -85,B 0,C 180,E1 -18853.289,E2 -18853.289} C_VEL
LIN {X 0,Y 250.127,Z 415.52,A -85,B 0,C 180,E1 -18857.596,E2 -18857.596} C_VEL
LIN {X 0,Y 249.412,Z 411.422,A -85,B 0,C 180,E1 -18861.689,E2 -18861.689} C_VEL
LIN {X 0,Y 249.121,Z 409.455,A -85,B 0,C 180,E1 -18863.847,E2 -18863.847} C_VEL
LIN {X 0,Y 249.046,Z 409.465,A -85,B 0,C 180,E1 -18867.847,E2 -18867.847} C_VEL
LIN {X 0,Y 249.094,Z 409.457,A -85,B 0,C 180,E1 -18871.338,E2 -18871.338} C_VEL
LIN {X 0,Y 249.16,Z 409.449,A -85,B 0,C 180,E1 -18874.969,E2 -18874.969} C_VEL
LIN {X 0,Y 249.12,Z 409.457,A -85,B 0,C 180,E1 -18880.212,E2 -18880.212} C_VEL
LIN {X 0,Y 249.251,Z 409.439,A -85,B 0,C 180,E1 -18883.622,E2 -18883.622} C_VEL
LIN {X 0,Y 249.253,Z 409.44,A -85,B 0,C 180,E1 -18888.616,E2 -18888.616} C_VEL
LIN {X 0,Y 249.463,Z 409.413,A -85,B 0,C 180,E1 -18891.902,E2 -18891.902} C_VEL
LIN {X 0,Y 249.301,Z 409.43,A -85,B 0,C 180,E1 -18895.148,E2 -18895.148} C_VEL
LIN {X 0,Y 249.683,Z 409.383,A -85,B 0,C 180,E1 -18898.387,E2 -18898.387} C_VEL
LIN {X 0,Y 249.683,Z 409.383,A -85,B 0,C 180,E1 -18901.613,E2 -18901.613} C_VEL
LIN {X 0,Y 249.457,Z 409.389,A -85,B 0,C 180,E1 -18906.806,E2 -18906.806} C_VEL
LIN {X 0,Y 249.398,Z 409.41,A -85,B 0,C 180,E1 -18909.734,E2 -18909.734} C_VEL
LIN {X 0,Y 249.21,Z 409.44,A -85,B 0,C 180,E1 -18914.703,E2 -18914.703} C_VEL
LIN {X 0,Y 249.147,Z 409.438,A -85,B 0,C 180,E1 -18918.077,E2 -18918.077} C_VEL
LIN {X 0,Y 249.096,Z 409.441,A -85,B 0,C 180,E1 -18921.517,E2 -18921.517} C_VEL
LIN {X 0,Y 249.139,Z 409.451,A -85,B 0,C 180,E1 -18925.481,E2 -18925.481} C_VEL
LIN {X 0,Y 249.081,Z 409.456,A -85,B 0,C 180,E1 -18928.988,E2 -18928.988} C_VEL
LIN {X 0,Y 249.038,Z 409.445,A -85,B 0,C 180,E1 -18932.425,E2 -18932.425} C_VEL
LIN {X 0,Y 249.055,Z 409.457,A -85,B 0,C 180,E1 -18936.341,E2 -18936.341} C_VEL
LIN {X 0,Y 249.013,Z 409.463,A -85,B 0,C 180,E1 -18940.477,E2 -18940.477} C_VEL
LIN {X 0,Y 249.014,Z 409.456,A -85,B 0,C 180,E1 -18944.877,E2 -18944.877} C_VEL
LIN {X 0,Y 249.025,Z 409.466,A -85,B 0,C 180,E1 -18947.362,E2 -18947.362} C_VEL
LIN {X 0,Y 249.05,Z 409.453,A -85,B 0,C 180,E1 -18952.199,E2 -18952.199} C_VEL
LIN {X 0,Y 249.05,Z 409.463,A -85,B 0,C 180,E1 -18955.637,E2 -18955.637} C_VEL
LIN {X 0,Y 249.058,Z 409.455,A -85,B 0,C 180,E1 -18959.471,E2 -18959.471} C_VEL
LIN {X 0,Y 249.079,Z 409.462,A -85,B 0,C 180,E1 -18963.16,E2 -18963.16} C_VEL
LIN {X 0,Y 249.085,Z 409.456,A -85,B 0,C 180,E1 -18966.73,E2 -18966.73} C_VEL
LIN {X 0,Y 249.116,Z 409.454,A -85,B 0,C 180,E1 -18970.209,E2 -18970.209} C_VEL
LIN {X 0,Y 249.247,Z 409.436,A -85,B 0,C 180,E1 -18973.619,E2 -18973.619} C_VEL
LIN {X 0,Y 249.127,Z 409.454,A -85,B 0,C 180,E1 -18976.954,E2 -18976.954} C_VEL
LIN {X 0,Y 248.956,Z 409.482,A -85,B 0,C 180,E1 -18980.245,E2 -18980.245} C_VEL
LIN {X 0,Y 249.036,Z 411.692,A -85,B 0,C 180,E1 -18983.515,E2 -18983.515} C_VEL
LIN {X 0,Y 248.955,Z 412.345,A -85,B 0,C 180,E1 -18984.428,E2 -18984.428} C_VEL
LIN {X 0,Y 253.645,Z 427.847,A -85,B 0,C 180,E1 -18985.938,E2 -18985.938} C_VEL
LIN {X 0,Y 256.725,Z 439.44,A -85,B 0,C 180,E1 -18987.31,E2 -18987.31} C_VEL
LIN {X 0,Y 258.835,Z 449.109,A -85,B 0,C 180,E1 -18988.636,E2 -18988.636} C_VEL
LIN {X 0,Y 259.463,Z 453.033,A -85,B 0,C 180,E1 -18989.221,E2 -18989.221} C_VEL
LIN {X 0,Y 257.732,Z 464.087,A -85,B 0,C 180,E1 -18990.778,E2 -18990.778} C_VEL
LIN {X 0,Y 255.649,Z 475.143,A -85,B 0,C 180,E1 -18992.754,E2 -18992.754} C_VEL
LIN {X 0,Y 253.792,Z 484.122,A -85,B 0,C 180,E1 -18994.762,E2 -18994.762} C_VEL
LIN {X 0,Y 251.892,Z 492.794,A -85,B 0,C 180,E1 -18997.21,E2 -18997.21} C_VEL
LIN {X 0,Y 250.367,Z 499.746,A -85,B 0,C 180,E1 -18999.693,E2 -18999.693} C_VEL
LIN {X 0,Y 249.205,Z 505.273,A -85,B 0,C 180,E1 -19002.208,E2 -19002.208} C_VEL
LIN {X 0,Y 248.292,Z 509.569,A -85,B 0,C 180,E1 -19004.755,E2 -19004.755} C_VEL
LIN {X 0,Y 247.83,Z 511.776,A -85,B 0,C 180,E1 -19006.47,E2 -19006.47} C_VEL
LIN {X 0,Y 247.418,Z 513.537,A -85,B 0,C 180,E1 -19008.204,E2 -19008.204} C_VEL
LIN {X 0,Y 247.156,Z 514.987,A -85,B 0,C 180,E1 -19010.22,E2 -19010.22} C_VEL
LIN {X 0,Y 247.051,Z 516.032,A -85,B 0,C 180,E1 -19013.466,E2 -19013.466} C_VEL
LIN {X 0,Y 247.154,Z 515.96,A -85,B 0,C 180,E1 -19015.244,E2 -19015.244} C_VEL
LIN {X 0,Y 247.649,Z 514.633,A -85,B 0,C 180,E1 -19018.388,E2 -19018.388} C_VEL
LIN {X 0,Y 248.268,Z 512.792,A -85,B 0,C 180,E1 -19020.629,E2 -19020.629} C_VEL
LIN {X 0,Y 249.265,Z 509.443,A -85,B 0,C 180,E1 -19023.349,E2 -19023.349} C_VEL
LIN {X 0,Y 250.644,Z 504.755,A -85,B 0,C 180,E1 -19026.07,E2 -19026.07} C_VEL
LIN {X 0,Y 252.433,Z 498.547,A -85,B 0,C 180,E1 -19028.781,E2 -19028.781} C_VEL
LIN {X 0,Y 254.282,Z 491.942,A -85,B 0,C 180,E1 -19031.022,E2 -19031.022} C_VEL
LIN {X 0,Y 256.397,Z 483.746,A -85,B 0,C 180,E1 -19033.251,E2 -19033.251} C_VEL
LIN {X 0,Y 258.614,Z 474.687,A -85,B 0,C 180,E1 -19035.227,E2 -19035.227} C_VEL
LIN {X 0,Y 260.741,Z 465.012,A -85,B 0,C 180,E1 -19036.924,E2 -19036.924} C_VEL
LIN {X 0,Y 262.024,Z 458.356,A -85,B 0,C 180,E1 -19037.891,E2 -19037.891} C_VEL
LIN {X 0,Y 261.528,Z 452.756,A -85,B 0,C 180,E1 -19038.796,E2 -19038.796} C_VEL
LIN {X 0,Y 259.199,Z 441.956,A -85,B 0,C 180,E1 -19040.488,E2 -19040.488} C_VEL
LIN {X 0,Y 255.738,Z 430.838,A -85,B 0,C 180,E1 -19042.104,E2 -19042.104} C_VEL
LIN {X 0,Y 251.244,Z 419.932,A -85,B 0,C 180,E1 -19043.61,E2 -19043.61} C_VEL
LIN {X 0,Y 249.097,Z 414.849,A -85,B 0,C 180,E1 -19044.242,E2 -19044.242} C_VEL
LIN {X 0,Y 249.024,Z 414.457,A -85,B 0,C 180,E1 -19044.362,E2 -19044.362} C_VEL
LIN {X 0,Y 249.176,Z 412.47,A -85,B 0,C 180,E1 -19047.788,E2 -19047.788} C_VEL
LIN {X 0,Y 249.201,Z 410.527,A -85,B 0,C 180,E1 -19051.352,E2 -19051.352} C_VEL
LIN {X 0,Y 249.067,Z 409.632,A -85,B 0,C 180,E1 -19053.162,E2 -19053.162} C_VEL
LIN {X 0,Y 249.146,Z 409.453,A -85,B 0,C 180,E1 -19054.968,E2 -19054.968} C_VEL
LIN {X 0,Y 249.145,Z 409.453,A -85,B 0,C 180,E1 -19058.561,E2 -19058.561} C_VEL
LIN {X 0,Y 249.225,Z 409.44,A -85,B 0,C 180,E1 -19063.621,E2 -19063.621} C_VEL
LIN {X 0,Y 249.235,Z 409.44,A -85,B 0,C 180,E1 -19068.616,E2 -19068.616} C_VEL
LIN {X 0,Y 249.464,Z 409.411,A -85,B 0,C 180,E1 -19071.902,E2 -19071.902} C_VEL
LIN {X 0,Y 249.421,Z 409.416,A -85,B 0,C 180,E1 -19076.77,E2 -19076.77} C_VEL
LIN {X 0,Y 249.718,Z 409.38,A -85,B 0,C 180,E1 -19080,E2 -19080} C_VEL
LIN {X 0,Y 249.45,Z 409.414,A -85,B 0,C 180,E1 -19083.23,E2 -19083.23} C_VEL
LIN {X 0,Y 249.464,Z 409.412,A -85,B 0,C 180,E1 -19088.098,E2 -19088.098} C_VEL
LIN {X 0,Y 249.236,Z 409.439,A -85,B 0,C 180,E1 -19091.384,E2 -19091.384} C_VEL
LIN {X 0,Y 249.226,Z 409.442,A -85,B 0,C 180,E1 -19096.379,E2 -19096.379} C_VEL
LIN {X 0,Y 249.127,Z 409.456,A -85,B 0,C 180,E1 -19101.515,E2 -19101.515} C_VEL
LIN {X 0,Y 249.122,Z 409.46,A -85,B 0,C 180,E1 -19105.487,E2 -19105.487} C_VEL
LIN {X 0,Y 249.058,Z 409.466,A -85,B 0,C 180,E1 -19108.991,E2 -19108.991} C_VEL
LIN {X 0,Y 249.03,Z 409.569,A -85,B 0,C 180,E1 -19110.959,E2 -19110.959} C_VEL
LIN {X 0,Y 249.617,Z 412.527,A -85,B 0,C 180,E1 -19115.271,E2 -19115.271} C_VEL
LIN {X 0,Y 249.863,Z 414.188,A -85,B 0,C 180,E1 -19117.416,E2 -19117.416} C_VEL
LIN {X 0,Y 249.421,Z 415.386,A -85,B 0,C 180,E1 -19118.737,E2 -19118.737} C_VEL
LIN {X 0,Y 246.968,Z 417.787,A -85,B 0,C 180,E1 -19120.882,E2 -19120.882} C_VEL
LIN {X 0,Y 244.861,Z 419.819,A -85,B 0,C 180,E1 -19122.622,E2 -19122.622} C_VEL
LIN {X 0,Y 244.042,Z 421.248,A -85,B 0,C 180,E1 -19123.969,E2 -19123.969} C_VEL
LIN {X 0,Y 244.025,Z 421.691,A -85,B 0,C 180,E1 -19124.424,E2 -19124.424} C_VEL
LIN {X 0,Y 244.764,Z 425.846,A -85,B 0,C 180,E1 -19128.674,E2 -19128.674} C_VEL
LIN {X 0,Y 245.174,Z 428.201,A -85,B 0,C 180,E1 -19130.908,E2 -19130.908} C_VEL
LIN {X 0,Y 245.08,Z 431.026,A -85,B 0,C 180,E1 -19133.412,E2 -19133.412} C_VEL
LIN {X 0,Y 243.846,Z 435.937,A -85,B 0,C 180,E1 -19137.411,E2 -19137.411} C_VEL
LIN {X 0,Y 243.717,Z 436.435,A -85,B 0,C 180,E1 -19137.807,E2 -19137.807} C_VEL
LIN {X 0,Y 244.588,Z 439.832,A -85,B 0,C 180,E1 -19138.125,E2 -19138.125} C_VEL
LIN {X 0,Y 247.645,Z 450.708,A -85,B 0,C 180,E1 -19139.325,E2 -19139.325} C_VEL
LIN {X 0,Y 249.917,Z 462.025,A -85,B 0,C 180,E1 -19140.665,E2 -19140.665} C_VEL
LIN {X 0,Y 251.386,Z 474.718,A -85,B 0,C 180,E1 -19142.344,E2 -19142.344} C_VEL
LIN {X 0,Y 251.669,Z 484.639,A -85,B 0,C 180,E1 -19143.82,E2 -19143.82} C_VEL
LIN {X 0,Y 251.232,Z 496.443,A -85,B 0,C 180,E1 -19145.854,E2 -19145.854} C_VEL
LIN {X 0,Y 249.046,Z 505.591,A -85,B 0,C 180,E1 -19147.61,E2 -19147.61} C_VEL
LIN {X 0,Y 246.448,Z 515.501,A -85,B 0,C 180,E1 -19149.992,E2 -19149.992} C_VEL
LIN {X 0,Y 244.824,Z 522.278,A -85,B 0,C 180,E1 -19152.029,E2 -19152.029} C_VEL
LIN {X 0,Y 242.996,Z 528.974,A -85,B 0,C 180,E1 -19154.486,E2 -19154.486} C_VEL
LIN {X 0,Y 241.428,Z 535.134,A -85,B 0,C 180,E1 -19157.393,E2 -19157.393} C_VEL
LIN {X 0,Y 240.618,Z 539.179,A -85,B 0,C 180,E1 -19159.91,E2 -19159.91} C_VEL
LIN {X 0,Y 240.082,Z 542.966,A -85,B 0,C 180,E1 -19163.279,E2 -19163.279} C_VEL
LIN {X 0,Y 239.989,Z 544.252,A -85,B 0,C 180,E1 -19164.963,E2 -19164.963} C_VEL
LIN {X 0,Y 240,Z 545.108,A -85,B 0,C 180,E1 -19166.646,E2 -19166.646} C_VEL
LIN {X 0,Y 240.032,Z 545.546,A -85,B 0,C 180,E1 -19168.325,E2 -19168.325} C_VEL
LIN {X 0,Y 240.103,Z 545.592,A -85,B 0,C 180,E1 -19170.003,E2 -19170.003} C_VEL
LIN {X 0,Y 240.053,Z 545.236,A -85,B 0,C 180,E1 -19171.681,E2 -19171.681} C_VEL
LIN {X 0,Y 240.036,Z 544.456,A -85,B 0,C 180,E1 -19173.36,E2 -19173.36} C_VEL
LIN {X 0,Y 240.035,Z 542.889,A -85,B 0,C 180,E1 -19175.441,E2 -19175.441} C_VEL
LIN {X 0,Y 240.307,Z 539.544,A -85,B 0,C 180,E1 -19178.412,E2 -19178.412} C_VEL
LIN {X 0,Y 240.858,Z 535.535,A -85,B 0,C 180,E1 -19180.936,E2 -19180.936} C_VEL
LIN {X 0,Y 241.958,Z 529.355,A -85,B 0,C 180,E1 -19183.868,E2 -19183.868} C_VEL
LIN {X 0,Y 243.391,Z 522.614,A -85,B 0,C 180,E1 -19186.355,E2 -19186.355} C_VEL
LIN {X 0,Y 244.911,Z 515.752,A -85,B 0,C 180,E1 -19188.403,E2 -19188.403} C_VEL
LIN {X 0,Y 246.567,Z 507.47,A -85,B 0,C 180,E1 -19190.439,E2 -19190.439} C_VEL
LIN {X 0,Y 248.487,Z 498.476,A -85,B 0,C 180,E1 -19192.231,E2 -19192.231} C_VEL
LIN {X 0,Y 249.332,Z 493.85,A -85,B 0,C 180,E1 -19193.026,E2 -19193.026} C_VEL
LIN {X 0,Y 249.147,Z 482.713,A -85,B 0,C 180,E1 -19194.812,E2 -19194.812} C_VEL
LIN {X 0,Y 248.493,Z 472.139,A -85,B 0,C 180,E1 -19196.228,E2 -19196.228} C_VEL
LIN {X 0,Y 246.954,Z 459.438,A -85,B 0,C 180,E1 -19197.652,E2 -19197.652} C_VEL
LIN {X 0,Y 244.492,Z 445.916,A -85,B 0,C 180,E1 -19198.895,E2 -19198.895} C_VEL
LIN {X 0,Y 242.804,Z 438.15,A -85,B 0,C 180,E1 -19199.48,E2 -19199.48} C_VEL
LIN {X 0,Y 244.123,Z 432.089,A -85,B 0,C 180,E1 -19204.153,E2 -19204.153} C_VEL
LIN {X 0,Y 244.89,Z 428.405,A -85,B 0,C 180,E1 -19207.065,E2 -19207.065} C_VEL
LIN {X 0,Y 244.76,Z 425.888,A -85,B 0,C 180,E1 -19209.179,E2 -19209.179} C_VEL
LIN {X 0,Y 243.92,Z 420.787,A -85,B 0,C 180,E1 -19213.753,E2 -19213.753} C_VEL
LIN {X 0,Y 243.003,Z 416.057,A -85,B 0,C 180,E1 -19218.302,E2 -19218.302} C_VEL
LIN {X 0,Y 242.206,Z 411.105,A -85,B 0,C 180,E1 -19223.499,E2 -19223.499} C_VEL
LIN {X 0,Y 242.046,Z 410.336,A -85,B 0,C 180,E1 -19224.499,E2 -19224.499} C_VEL
LIN {X 0,Y 241.982,Z 410.348,A -85,B 0,C 180,E1 -19228.481,E2 -19228.481} C_VEL
LIN {X 0,Y 242.011,Z 410.342,A -85,B 0,C 180,E1 -19232.313,E2 -19232.313} C_VEL
LIN {X 0,Y 242.066,Z 410.332,A -85,B 0,C 180,E1 -19236.017,E2 -19236.017} C_VEL
LIN {X 0,Y 242.047,Z 410.336,A -85,B 0,C 180,E1 -19239.609,E2 -19239.609} C_VEL
LIN {X 0,Y 242.173,Z 410.321,A -85,B 0,C 180,E1 -19243.279,E2 -19243.279} C_VEL
LIN {X 0,Y 242.189,Z 410.322,A -85,B 0,C 180,E1 -19248.28,E2 -19248.28} C_VEL
LIN {X 0,Y 242.409,Z 410.291,A -85,B 0,C 180,E1 -19251.665,E2 -19251.665} C_VEL
LIN {X 0,Y 242.262,Z 410.307,A -85,B 0,C 180,E1 -19255.007,E2 -19255.007} C_VEL
LIN {X 0,Y 242.643,Z 410.26,A -85,B 0,C 180,E1 -19258.34,E2 -19258.34} C_VEL
LIN {X 0,Y 242.643,Z 410.26,A -85,B 0,C 180,E1 -19261.66,E2 -19261.66} C_VEL
LIN {X 0,Y 242.433,Z 410.263,A -85,B 0,C 180,E1 -19266.785,E2 -19266.785} C_VEL
LIN {X 0,Y 242.323,Z 410.293,A -85,B 0,C 180,E1 -19270.021,E2 -19270.021} C_VEL
LIN {X 0,Y 242.173,Z 410.317,A -85,B 0,C 180,E1 -19275.14,E2 -19275.14} C_VEL
LIN {X 0,Y 242.081,Z 410.315,A -85,B 0,C 180,E1 -19278.623,E2 -19278.623} C_VEL
LIN {X 0,Y 242.022,Z 410.328,A -85,B 0,C 180,E1 -19282.179,E2 -19282.179} C_VEL
LIN {X 0,Y 242.075,Z 410.332,A -85,B 0,C 180,E1 -19285.837,E2 -19285.837} C_VEL
LIN {X 0,Y 242.015,Z 410.333,A -85,B 0,C 180,E1 -19289.582,E2 -19289.582} C_VEL
LIN {X 0,Y 241.988,Z 410.325,A -85,B 0,C 180,E1 -19293.491,E2 -19293.491} C_VEL
LIN {X 0,Y 241.997,Z 410.342,A -85,B 0,C 180,E1 -19297.58,E2 -19297.58} C_VEL
LIN {X 0,Y 241.946,Z 410.338,A -85,B 0,C 180,E1 -19301.92,E2 -19301.92} C_VEL
LIN {X 0,Y 241.944,Z 410.343,A -85,B 0,C 180,E1 -19306.569,E2 -19306.569} C_VEL
LIN {X 0,Y 241.963,Z 410.342,A -85,B 0,C 180,E1 -19310.279,E2 -19310.279} C_VEL
LIN {X 0,Y 241.994,Z 410.338,A -85,B 0,C 180,E1 -19314.487,E2 -19314.487} C_VEL
LIN {X 0,Y 241.981,Z 410.343,A -85,B 0,C 180,E1 -19318.478,E2 -19318.478} C_VEL
LIN {X 0,Y 242.014,Z 410.34,A -85,B 0,C 180,E1 -19322.31,E2 -19322.31} C_VEL
LIN {X 0,Y 242.063,Z 410.329,A -85,B 0,C 180,E1 -19326.014,E2 -19326.014} C_VEL
LIN {X 0,Y 242.043,Z 410.334,A -85,B 0,C 180,E1 -19329.605,E2 -19329.605} C_VEL
LIN {X 0,Y 242.168,Z 410.318,A -85,B 0,C 180,E1 -19333.276,E2 -19333.276} C_VEL
LIN {X 0,Y 242.095,Z 410.33,A -85,B 0,C 180,E1 -19336.568,E2 -19336.568} C_VEL
LIN {X 0,Y 241.914,Z 410.352,A -85,B 0,C 180,E1 -19339.958,E2 -19339.958} C_VEL
LIN {X 0,Y 242.008,Z 412.8,A -85,B 0,C 180,E1 -19343.64,E2 -19343.64} C_VEL
LIN {X 0,Y 246.543,Z 427.566,A -85,B 0,C 180,E1 -19345.13,E2 -19345.13} C_VEL
LIN {X 0,Y 249.654,Z 439.046,A -85,B 0,C 180,E1 -19346.527,E2 -19346.527} C_VEL
LIN {X 0,Y 252.079,Z 450.005,A -85,B 0,C 180,E1 -19348.085,E2 -19348.085} C_VEL
LIN {X 0,Y 252.735,Z 454.676,A -85,B 0,C 180,E1 -19348.802,E2 -19348.802} C_VEL
LIN {X 0,Y 250.904,Z 465.47,A -85,B 0,C 180,E1 -19350.398,E2 -19350.398} C_VEL
LIN {X 0,Y 248.757,Z 476.37,A -85,B 0,C 180,E1 -19352.426,E2 -19352.426} C_VEL
LIN {X 0,Y 246.773,Z 485.575,A -85,B 0,C 180,E1 -19354.593,E2 -19354.593} C_VEL
LIN {X 0,Y 244.901,Z 493.73,A -85,B 0,C 180,E1 -19357.002,E2 -19357.002} C_VEL
LIN {X 0,Y 243.311,Z 500.601,A -85,B 0,C 180,E1 -19359.557,E2 -19359.557} C_VEL
LIN {X 0,Y 242.309,Z 505.195,A -85,B 0,C 180,E1 -19361.711,E2 -19361.711} C_VEL
LIN {X 0,Y 241.331,Z 509.608,A -85,B 0,C 180,E1 -19364.328,E2 -19364.328} C_VEL
LIN {X 0,Y 240.59,Z 512.891,A -85,B 0,C 180,E1 -19366.981,E2 -19366.981} C_VEL
LIN {X 0,Y 240.243,Z 514.484,A -85,B 0,C 180,E1 -19368.767,E2 -19368.767} C_VEL
LIN {X 0,Y 240.029,Z 515.598,A -85,B 0,C 180,E1 -19370.566,E2 -19370.566} C_VEL
LIN {X 0,Y 239.941,Z 516.288,A -85,B 0,C 180,E1 -19372.378,E2 -19372.378} C_VEL
LIN {X 0,Y 240.026,Z 516.456,A -85,B 0,C 180,E1 -19374.813,E2 -19374.813} C_VEL
LIN {X 0,Y 240.442,Z 515.528,A -85,B 0,C 180,E1 -19377.879,E2 -19377.879} C_VEL
LIN {X 0,Y 240.914,Z 514.287,A -85,B 0,C 180,E1 -19379.727,E2 -19379.727} C_VEL
LIN {X 0,Y 241.862,Z 511.406,A -85,B 0,C 180,E1 -19382.576,E2 -19382.576} C_VEL
LIN {X 0,Y 243.116,Z 507.394,A -85,B 0,C 180,E1 -19385.317,E2 -19385.317} C_VEL
LIN {X 0,Y 244.862,Z 501.894,A -85,B 0,C 180,E1 -19388.099,E2 -19388.099} C_VEL
LIN {X 0,Y 246.975,Z 494.63,A -85,B 0,C 180,E1 -19390.876,E2 -19390.876} C_VEL
LIN {X 0,Y 249.072,Z 487.189,A -85,B 0,C 180,E1 -19393.116,E2 -19393.116} C_VEL
LIN {X 0,Y 251.476,Z 478.057,A -85,B 0,C 180,E1 -19395.315,E2 -19395.315} C_VEL
LIN {X 0,Y 253.825,Z 468.155,A -85,B 0,C 180,E1 -19397.195,E2 -19397.195} C_VEL
LIN {X 0,Y 255.563,Z 459.887,A -85,B 0,C 180,E1 -19398.483,E2 -19398.483} C_VEL
LIN {X 0,Y 255.42,Z 456.526,A -85,B 0,C 180,E1 -19399.048,E2 -19399.048} C_VEL
LIN {X 0,Y 253.42,Z 445.961,A -85,B 0,C 180,E1 -19400.832,E2 -19400.832} C_VEL
LIN {X 0,Y 250.174,Z 434.665,A -85,B 0,C 180,E1 -19402.591,E2 -19402.591} C_VEL
LIN {X 0,Y 245.384,Z 422.394,A -85,B 0,C 180,E1 -19404.4,E2 -19404.4} C_VEL
LIN {X 0,Y 242.254,Z 415.816,A -85,B 0,C 180,E1 -19405.359,E2 -19405.359} C_VEL
LIN {X 0,Y 242.109,Z 414.973,A -85,B 0,C 180,E1 -19405.525,E2 -19405.525} C_VEL
LIN {X 0,Y 242.17,Z 413.329,A -85,B 0,C 180,E1 -19408.508,E2 -19408.508} C_VEL
LIN {X 0,Y 242.144,Z 411.36,A -85,B 0,C 180,E1 -19412.33,E2 -19412.33} C_VEL
LIN {X 0,Y 242.078,Z 410.47,A -85,B 0,C 180,E1 -19414.184,E2 -19414.184} C_VEL
LIN {X 0,Y 242.074,Z 410.332,A -85,B 0,C 180,E1 -19418.274,E2 -19418.274} C_VEL
LIN {X 0,Y 242.147,Z 410.323,A -85,B 0,C 180,E1 -19423.277,E2 -19423.277} C_VEL
LIN {X 0,Y 242.169,Z 410.321,A -85,B 0,C 180,E1 -19428.279,E2 -19428.279} C_VEL
LIN {X 0,Y 242.411,Z 410.29,A -85,B 0,C 180,E1 -19431.665,E2 -19431.665} C_VEL
LIN {X 0,Y 242.247,Z 410.311,A -85,B 0,C 180,E1 -19435.007,E2 -19435.007} C_VEL
LIN {X 0,Y 242.62,Z 410.264,A -85,B 0,C 180,E1 -19438.34,E2 -19438.34} C_VEL
LIN {X 0,Y 242.629,Z 410.264,A -85,B 0,C 180,E1 -19441.66,E2 -19441.66} C_VEL
LIN {X 0,Y 242.416,Z 410.29,A -85,B 0,C 180,E1 -19446.659,E2 -19446.659} C_VEL
LIN {X 0,Y 242.297,Z 410.305,A -85,B 0,C 180,E1 -19450.023,E2 -19450.023} C_VEL
LIN {X 0,Y 242.15,Z 410.323,A -85,B 0,C 180,E1 -19455.142,E2 -19455.142} C_VEL
LIN {X 0,Y 242.077,Z 410.332,A -85,B 0,C 180,E1 -19458.624,E2 -19458.624} C_VEL
LIN {X 0,Y 242.06,Z 410.336,A -85,B 0,C 180,E1 -19462.176,E2 -19462.176} C_VEL
LIN {X 0,Y 242.052,Z 410.34,A -85,B 0,C 180,E1 -19465.84,E2 -19465.84} C_VEL
LIN {X 0,Y 242.012,Z 410.393,A -85,B 0,C 180,E1 -19469.583,E2 -19469.583} C_VEL
LIN {X 0,Y 242.411,Z 412.827,A -85,B 0,C 180,E1 -19473.426,E2 -19473.426} C_VEL
LIN {X 0,Y 242.947,Z 415.725,A -85,B 0,C 180,E1 -19477.409,E2 -19477.409} C_VEL
LIN {X 0,Y 243.577,Z 419.135,A -85,B 0,C 180,E1 -19481.577,E2 -19481.577} C_VEL
LIN {X 0,Y 244.025,Z 421.691,A -85,B 0,C 180,E1 -19484.424,E2 -19484.424} C_VEL
LIN {X 0,Y 243.57,Z 423.099,A -85,B 0,C 180,E1 -19485.766,E2 -19485.766} C_VEL
LIN {X 0,Y 241.113,Z 425.762,A -85,B 0,C 180,E1 -19487.947,E2 -19487.947} C_VEL
LIN {X 0,Y 239.013,Z 427.975,A -85,B 0,C 180,E1 -19489.717,E2 -19489.717} C_VEL
LIN {X 0,Y 238.205,Z 429.569,A -85,B 0,C 180,E1 -19491.086,E2 -19491.086} C_VEL
LIN {X 0,Y 238.193,Z 430.072,A -85,B 0,C 180,E1 -19491.55,E2 -19491.55} C_VEL
LIN {X 0,Y 237.888,Z 432.59,A -85,B 0,C 180,E1 -19493.786,E2 -19493.786} C_VEL
LIN {X 0,Y 237.021,Z 435.929,A -85,B 0,C 180,E1 -19496.611,E2 -19496.611} C_VEL
LIN {X 0,Y 237.867,Z 439.261,A -85,B 0,C 180,E1 -19496.945,E2 -19496.945} C_VEL
LIN {X 0,Y 241.164,Z 450.662,A -85,B 0,C 180,E1 -19498.294,E2 -19498.294} C_VEL
LIN {X 0,Y 243.367,Z 461.663,A -85,B 0,C 180,E1 -19499.676,E2 -19499.676} C_VEL
LIN {X 0,Y 244.82,Z 474.024,A -85,B 0,C 180,E1 -19501.387,E2 -19501.387} C_VEL
LIN {X 0,Y 245.176,Z 484.87,A -85,B 0,C 180,E1 -19503.071,E2 -19503.071} C_VEL
LIN {X 0,Y 244.673,Z 495.383,A -85,B 0,C 180,E1 -19504.937,E2 -19504.937} C_VEL
LIN {X 0,Y 244.09,Z 499.7,A -85,B 0,C 180,E1 -19505.781,E2 -19505.781} C_VEL
LIN {X 0,Y 241.509,Z 509.083,A -85,B 0,C 180,E1 -19507.775,E2 -19507.775} C_VEL
LIN {X 0,Y 238.984,Z 518.167,A -85,B 0,C 180,E1 -19510.229,E2 -19510.229} C_VEL
LIN {X 0,Y 237.682,Z 523.319,A -85,B 0,C 180,E1 -19511.916,E2 -19511.916} C_VEL
LIN {X 0,Y 235.85,Z 529.713,A -85,B 0,C 180,E1 -19514.447,E2 -19514.447} C_VEL
LIN {X 0,Y 234.446,Z 534.837,A -85,B 0,C 180,E1 -19517.011,E2 -19517.011} C_VEL
LIN {X 0,Y 233.587,Z 538.846,A -85,B 0,C 180,E1 -19519.603,E2 -19519.603} C_VEL
LIN {X 0,Y 233.227,Z 540.93,A -85,B 0,C 180,E1 -19521.338,E2 -19521.338} C_VEL
LIN {X 0,Y 232.913,Z 543.813,A -85,B 0,C 180,E1 -19524.722,E2 -19524.722} C_VEL
LIN {X 0,Y 232.917,Z 544.697,A -85,B 0,C 180,E1 -19526.544,E2 -19526.544} C_VEL
LIN {X 0,Y 232.96,Z 545.121,A -85,B 0,C 180,E1 -19528.275,E2 -19528.275} C_VEL
LIN {X 0,Y 233.027,Z 545.152,A -85,B 0,C 180,E1 -19530.003,E2 -19530.003} C_VEL
LIN {X 0,Y 232.981,Z 544.782,A -85,B 0,C 180,E1 -19531.732,E2 -19531.732} C_VEL
LIN {X 0,Y 232.95,Z 543.97,A -85,B 0,C 180,E1 -19533.463,E2 -19533.463} C_VEL
LIN {X 0,Y 232.956,Z 542.568,A -85,B 0,C 180,E1 -19535.391,E2 -19535.391} C_VEL
LIN {X 0,Y 233.255,Z 539,A -85,B 0,C 180,E1 -19538.668,E2 -19538.668} C_VEL
LIN {X 0,Y 233.866,Z 534.956,A -85,B 0,C 180,E1 -19541.267,E2 -19541.267} C_VEL
LIN {X 0,Y 235.046,Z 528.721,A -85,B 0,C 180,E1 -19544.284,E2 -19544.284} C_VEL
LIN {X 0,Y 236.547,Z 521.93,A -85,B 0,C 180,E1 -19546.842,E2 -19546.842} C_VEL
LIN {X 0,Y 237.83,Z 516.512,A -85,B 0,C 180,E1 -19548.525,E2 -19548.525} C_VEL
LIN {X 0,Y 239.49,Z 508.459,A -85,B 0,C 180,E1 -19550.622,E2 -19550.622} C_VEL
LIN {X 0,Y 241.65,Z 498.671,A -85,B 0,C 180,E1 -19552.669,E2 -19552.669} C_VEL
LIN {X 0,Y 242.478,Z 494.1,A -85,B 0,C 180,E1 -19553.489,E2 -19553.489} C_VEL
LIN {X 0,Y 242.372,Z 483.435,A -85,B 0,C 180,E1 -19555.283,E2 -19555.283} C_VEL
LIN {X 0,Y 241.79,Z 473.054,A -85,B 0,C 180,E1 -19556.752,E2 -19556.752} C_VEL
LIN {X 0,Y 240.416,Z 461.107,A -85,B 0,C 180,E1 -19558.181,E2 -19558.181} C_VEL
LIN {X 0,Y 238.065,Z 447.639,A -85,B 0,C 180,E1 -19559.504,E2 -19559.504} C_VEL
LIN {X 0,Y 235.943,Z 437.713,A -85,B 0,C 180,E1 -19560.33,E2 -19560.33} C_VEL
LIN {X 0,Y 237.412,Z 431.531,A -85,B 0,C 180,E1 -19565.26,E2 -19565.26} C_VEL
LIN {X 0,Y 237.844,Z 429.307,A -85,B 0,C 180,E1 -19567.077,E2 -19567.077} C_VEL
LIN {X 0,Y 237.637,Z 426.255,A -85,B 0,C 180,E1 -19569.741,E2 -19569.741} C_VEL
LIN {X 0,Y 237.085,Z 422.731,A -85,B 0,C 180,E1 -19572.988,E2 -19572.988} C_VEL
LIN {X 0,Y 236.318,Z 418.767,A -85,B 0,C 180,E1 -19576.842,E2 -19576.842} C_VEL
LIN {X 0,Y 235.522,Z 414.59,A -85,B 0,C 180,E1 -19581.197,E2 -19581.197} C_VEL
LIN {X 0,Y 234.98,Z 411.236,A -85,B 0,C 180,E1 -19584.966,E2 -19584.966} C_VEL
LIN {X 0,Y 234.931,Z 411.224,A -85,B 0,C 180,E1 -19589.432,E2 -19589.432} C_VEL
LIN {X 0,Y 235.003,Z 411.211,A -85,B 0,C 180,E1 -19593.795,E2 -19593.795} C_VEL
LIN {X 0,Y 235.021,Z 411.213,A -85,B 0,C 180,E1 -19598.971,E2 -19598.971} C_VEL
LIN {X 0,Y 235.106,Z 411.202,A -85,B 0,C 180,E1 -19603.06,E2 -19603.06} C_VEL
LIN {X 0,Y 235.123,Z 411.201,A -85,B 0,C 180,E1 -19607.922,E2 -19607.922} C_VEL
LIN {X 0,Y 235.34,Z 411.171,A -85,B 0,C 180,E1 -19611.413,E2 -19611.413} C_VEL
LIN {X 0,Y 235.382,Z 411.165,A -85,B 0,C 180,E1 -19613.141,E2 -19613.141} C_VEL
LIN {X 0,Y 235.603,Z 411.138,A -85,B 0,C 180,E1 -19618.29,E2 -19618.29} C_VEL
LIN {X 0,Y 235.603,Z 411.137,A -85,B 0,C 180,E1 -19621.709,E2 -19621.709} C_VEL
LIN {X 0,Y 235.412,Z 411.136,A -85,B 0,C 180,E1 -19626.858,E2 -19626.858} C_VEL
LIN {X 0,Y 235.247,Z 411.177,A -85,B 0,C 180,E1 -19630.326,E2 -19630.326} C_VEL
LIN {X 0,Y 235.121,Z 411.196,A -85,B 0,C 180,E1 -19635.606,E2 -19635.606} C_VEL
LIN {X 0,Y 235.017,Z 411.192,A -85,B 0,C 180,E1 -19639.205,E2 -19639.205} C_VEL
LIN {X 0,Y 234.97,Z 411.206,A -85,B 0,C 180,E1 -19642.882,E2 -19642.882} C_VEL
LIN {X 0,Y 234.976,Z 411.214,A -85,B 0,C 180,E1 -19646.656,E2 -19646.656} C_VEL
LIN {X 0,Y 234.93,Z 411.211,A -85,B 0,C 180,E1 -19650.568,E2 -19650.568} C_VEL
LIN {X 0,Y 234.938,Z 411.208,A -85,B 0,C 180,E1 -19654.637,E2 -19654.637} C_VEL
LIN {X 0,Y 234.95,Z 411.219,A -85,B 0,C 180,E1 -19658.943,E2 -19658.943} C_VEL
LIN {X 0,Y 234.897,Z 411.21,A -85,B 0,C 180,E1 -19663.484,E2 -19663.484} C_VEL
LIN {X 0,Y 234.897,Z 411.221,A -85,B 0,C 180,E1 -19666.513,E2 -19666.513} C_VEL
LIN {X 0,Y 234.925,Z 411.215,A -85,B 0,C 180,E1 -19671.077,E2 -19671.077} C_VEL
LIN {X 0,Y 234.936,Z 411.223,A -85,B 0,C 180,E1 -19675.36,E2 -19675.36} C_VEL
LIN {X 0,Y 234.938,Z 411.213,A -85,B 0,C 180,E1 -19679.43,E2 -19679.43} C_VEL
LIN {X 0,Y 235,Z 411.215,A -85,B 0,C 180,E1 -19683.791,E2 -19683.791} C_VEL
LIN {X 0,Y 235.017,Z 411.212,A -85,B 0,C 180,E1 -19688.967,E2 -19688.967} C_VEL
LIN {X 0,Y 235.101,Z 411.2,A -85,B 0,C 180,E1 -19693.057,E2 -19693.057} C_VEL
LIN {X 0,Y 235.054,Z 411.207,A -85,B 0,C 180,E1 -19696.158,E2 -19696.158} C_VEL
LIN {X 0,Y 234.873,Z 411.23,A -85,B 0,C 180,E1 -19699.654,E2 -19699.654} C_VEL
LIN {X 0,Y 234.978,Z 413.245,A -85,B 0,C 180,E1 -19702.802,E2 -19702.802} C_VEL
LIN {X 0,Y 239.166,Z 426.029,A -85,B 0,C 180,E1 -19704.149,E2 -19704.149} C_VEL
LIN {X 0,Y 242.538,Z 438.451,A -85,B 0,C 180,E1 -19705.68,E2 -19705.68} C_VEL
LIN {X 0,Y 245.109,Z 449.813,A -85,B 0,C 180,E1 -19707.326,E2 -19707.326} C_VEL
LIN {X 0,Y 245.994,Z 456.25,A -85,B 0,C 180,E1 -19708.36,E2 -19708.36} C_VEL
LIN {X 0,Y 243.861,Z 468.054,A -85,B 0,C 180,E1 -19710.203,E2 -19710.203} C_VEL
LIN {X 0,Y 241.86,Z 477.582,A -85,B 0,C 180,E1 -19712.078,E2 -19712.078} C_VEL
LIN {X 0,Y 239.683,Z 487.227,A -85,B 0,C 180,E1 -19714.475,E2 -19714.475} C_VEL
LIN {X 0,Y 237.913,Z 494.668,A -85,B 0,C 180,E1 -19716.783,E2 -19716.783} C_VEL
LIN {X 0,Y 236.273,Z 501.446,A -85,B 0,C 180,E1 -19719.412,E2 -19719.412} C_VEL
LIN {X 0,Y 235.044,Z 506.777,A -85,B 0,C 180,E1 -19722.078,E2 -19722.078} C_VEL
LIN {X 0,Y 234.111,Z 510.901,A -85,B 0,C 180,E1 -19724.78,E2 -19724.78} C_VEL
LIN {X 0,Y 233.393,Z 513.927,A -85,B 0,C 180,E1 -19727.521,E2 -19727.521} C_VEL
LIN {X 0,Y 232.925,Z 516.103,A -85,B 0,C 180,E1 -19730.714,E2 -19730.714} C_VEL
LIN {X 0,Y 232.846,Z 516.839,A -85,B 0,C 180,E1 -19733.098,E2 -19733.098} C_VEL
LIN {X 0,Y 232.969,Z 516.879,A -85,B 0,C 180,E1 -19735.175,E2 -19735.175} C_VEL
LIN {X 0,Y 233.2,Z 516.494,A -85,B 0,C 180,E1 -19736.872,E2 -19736.872} C_VEL
LIN {X 0,Y 233.734,Z 515.241,A -85,B 0,C 180,E1 -19739.31,E2 -19739.31} C_VEL
LIN {X 0,Y 234.793,Z 512.266,A -85,B 0,C 180,E1 -19742.597,E2 -19742.597} C_VEL
LIN {X 0,Y 236.085,Z 508.31,A -85,B 0,C 180,E1 -19745.48,E2 -19745.48} C_VEL
LIN {X 0,Y 237.902,Z 502.952,A -85,B 0,C 180,E1 -19748.338,E2 -19748.338} C_VEL
LIN {X 0,Y 239.686,Z 497.214,A -85,B 0,C 180,E1 -19750.718,E2 -19750.718} C_VEL
LIN {X 0,Y 241.797,Z 490.393,A -85,B 0,C 180,E1 -19752.981,E2 -19752.981} C_VEL
LIN {X 0,Y 244.3,Z 481.269,A -85,B 0,C 180,E1 -19755.393,E2 -19755.393} C_VEL
LIN {X 0,Y 246.836,Z 471.76,A -85,B 0,C 180,E1 -19757.368,E2 -19757.368} C_VEL
LIN {X 0,Y 249.034,Z 461.994,A -85,B 0,C 180,E1 -19759.012,E2 -19759.012} C_VEL
LIN {X 0,Y 249.091,Z 458.914,A -85,B 0,C 180,E1 -19759.539,E2 -19759.539} C_VEL
LIN {X 0,Y 247.387,Z 449.023,A -85,B 0,C 180,E1 -19761.318,E2 -19761.318} C_VEL
LIN {X 0,Y 244.863,Z 439.385,A -85,B 0,C 180,E1 -19762.934,E2 -19762.934} C_VEL
LIN {X 0,Y 240.449,Z 427.293,A -85,B 0,C 180,E1 -19764.887,E2 -19764.887} C_VEL
LIN {X 0,Y 236.607,Z 419.144,A -85,B 0,C 180,E1 -19766.187,E2 -19766.187} C_VEL
LIN {X 0,Y 235.219,Z 416.041,A -85,B 0,C 180,E1 -19766.644,E2 -19766.644} C_VEL
LIN {X 0,Y 235.138,Z 415.541,A -85,B 0,C 180,E1 -19766.72,E2 -19766.72} C_VEL
LIN {X 0,Y 235.2,Z 413.806,A -85,B 0,C 180,E1 -19770.051,E2 -19770.051} C_VEL
LIN {X 0,Y 235.099,Z 412.038,A -85,B 0,C 180,E1 -19773.732,E2 -19773.732} C_VEL
LIN {X 0,Y 235.01,Z 411.368,A -85,B 0,C 180,E1 -19775.249,E2 -19775.249} C_VEL
LIN {X 0,Y 235.035,Z 411.21,A -85,B 0,C 180,E1 -19778.972,E2 -19778.972} C_VEL
LIN {X 0,Y 235.1,Z 411.202,A -85,B 0,C 180,E1 -19783.042,E2 -19783.042} C_VEL
LIN {X 0,Y 235.101,Z 411.199,A -85,B 0,C 180,E1 -19787.921,E2 -19787.921} C_VEL
LIN {X 0,Y 235.36,Z 411.17,A -85,B 0,C 180,E1 -19791.414,E2 -19791.414} C_VEL
LIN {X 0,Y 235.388,Z 411.158,A -85,B 0,C 180,E1 -19793.141,E2 -19793.141} C_VEL
LIN {X 0,Y 235.58,Z 411.141,A -85,B 0,C 180,E1 -19798.291,E2 -19798.291} C_VEL
LIN {X 0,Y 235.589,Z 411.14,A -85,B 0,C 180,E1 -19801.71,E2 -19801.71} C_VEL
LIN {X 0,Y 235.387,Z 411.165,A -85,B 0,C 180,E1 -19806.859,E2 -19806.859} C_VEL
LIN {X 0,Y 235.221,Z 411.185,A -85,B 0,C 180,E1 -19810.327,E2 -19810.327} C_VEL
LIN {X 0,Y 235.097,Z 411.201,A -85,B 0,C 180,E1 -19815.608,E2 -19815.608} C_VEL
LIN {X 0,Y 235.02,Z 411.212,A -85,B 0,C 180,E1 -19819.205,E2 -19819.205} C_VEL
LIN {X 0,Y 234.99,Z 411.219,A -85,B 0,C 180,E1 -19822.88,E2 -19822.88} C_VEL
LIN {X 0,Y 234.953,Z 411.224,A -85,B 0,C 180,E1 -19826.66,E2 -19826.66} C_VEL
LIN {X 0,Y 234.991,Z 411.523,A -85,B 0,C 180,E1 -19828.589,E2 -19828.589} C_VEL
LIN {X 0,Y 235.421,Z 413.839,A -85,B 0,C 180,E1 -19832.504,E2 -19832.504} C_VEL
LIN {X 0,Y 235.908,Z 416.636,A -85,B 0,C 180,E1 -19836.572,E2 -19836.572} C_VEL
LIN {X 0,Y 236.49,Z 419.959,A -85,B 0,C 180,E1 -19840.829,E2 -19840.829} C_VEL
LIN {X 0,Y 237.225,Z 423.884,A -85,B 0,C 180,E1 -19845.318,E2 -19845.318} C_VEL
